DATA_BLOCK "iPar_Data_Bridge"	// DB 1920
TITLE = Vorlage Datenbaustein zur Ablage der iParameter für FB37
//Template data block used in combination with FB37
//
AUTHOR : JPR
FAMILY : WAGOiPar
NAME : iParUDL4
VERSION : 5.1
  STRUCT
   versionInfo_1 : INT  := 37;	//version info main
   versionInfo_2 : WORD  := W#16#501;	//version info release
   chkInfoData : WORD ;	//check info data
   fctReqTimeout : INT  := 6000;	//function request timeout (default 6000; av.cycle plc 5 ms - timeout 30 s)
   maxModules : INT  := 1;	//amount PROFIsafe modules FB41
   type_module_1 : INT ;	//type module 1 (661/662/663/666/667/669)
   adr_module_1 : INT ;	//I/O address module 1
   bussystem_mod_1 : INT ;	//used bussystem module 1 (0 = DP / 1 = PN)
   type_module_2 : INT ;	//type module 2 (661/662/663/666/667/669)
   adr_module_2 : INT ;	//I/O address module 2
   bussystem_mod_2 : INT ;	//used bussystem module 2 (0 = DP / 1 = PN)
   type_module_3 : INT ;	//type module 3 (661/662/663/666/667/669)
   adr_module_3 : INT ;	//I/O address module 3
   bussystem_mod_3 : INT ;	//used bussystem module 3 (0 = DP / 1 = PN)
   type_module_4 : INT ;	//type module 4 (661/662/663/666/667/669)
   adr_module_4 : INT ;	//I/O address module 4
   bussystem_mod_4 : INT ;	//used bussystem module 4 (0 = DP / 1 = PN)
   spare_34 : WORD ;
   spare_36 : WORD ;
   spare_38 : WORD ;
   spare_40 : WORD ;
   spare_42 : WORD ;
   spare_44 : WORD ;
   spare_46 : WORD ;
   spare_48 : WORD ;
   spare_50 : WORD ;
   spare_52 : WORD ;
   spare_54 : WORD ;
   spare_56 : WORD ;
   spare_58 : WORD ;
   spare_60 : WORD ;
   spare_62 : WORD ;
   spare_64 : WORD ;
   spare_66 : WORD ;
   spare_68 : WORD ;
   spare_70 : WORD ;
   spare_72 : WORD ;
   spare_74 : WORD ;
   spare_76 : WORD ;
   spare_78 : WORD ;
   spare_80 : WORD ;
   resFctReq_ok : DWORD ;	//response function request ok - "bit per module"
   resFctReq_error : DWORD ;	//response function request error - "bit per module"
   startupDate : DATE ;	//startup date application slave
   startupTime : TIME_OF_DAY ;	//startup time application slave
   slaveConfigInfo : DWORD ;	//info available PROFIsafe modules at slave
   QBAD_moduleActive : DWORD ;	//info QBAD at PROFIsafe module active
   ACK_REQ_moduleActive : DWORD ;	//info ACK_REQ at PROFIsafe module active
   READ_DIAG_REQ_module : DWORD ;	//info READ_DIAG_REQ at PROFIsafe module active
   init_fb_done : DWORD ;	//info init FB done
   check_cfg_done : DWORD ;	//info check cfg done
   upload_done : DWORD ;	//info upload slave done
   download_done : DWORD ;	//info download slave done
   compare_done : DWORD ;	//info compare slave done
   actDateCyle : DATE ;	//actual system date of cycle
   actTimeCyle : TIME_OF_DAY ;	//actual system time of cycle
   cmdCtrl_FB37 : WORD ;	//cmd / ctrl information FB37
   comCountStart_1 : WORD ;	//comCountStart indication 1
   mod_type_1 : WORD ;	//module type 1
   mod_version_1 : WORD ;	//module version 1
   spare_146 : WORD ;
   spare_148 : WORD ;
   upl_date_mod_1 : DATE ;	//upload date module 1
   upl_time_mod_1 : TIME_OF_DAY ;	//upload time module 1
   dnl_date_mod_1 : DATE ;	//download date module 1
   dnl_time_mod_1 : TIME_OF_DAY ;	//download time module 1
   cmp_date_mod_1 : DATE ;	//compare date module 1
   cmp_time_mod_1 : TIME_OF_DAY ;	//compare time module 1
   dsv_info_mod_1 : WORD ;	//dataset info module 1
   data_0_mod_1 : WORD ;	//data 0 - 1 module 1
   data_2_mod_1 : WORD ;	//data 2 - 3 module 1
   data_4_mod_1 : WORD ;	//data 4 - 5 module 1
   data_6_mod_1 : WORD ;	//data 6 - 7 module 1
   data_8_mod_1 : WORD ;	//data 8 - 9 module 1
   data_10_mod_1 : WORD ;	//data 10 - 11 module 1
   data_12_mod_1 : WORD ;	//data 12 - 13 module 1
   data_14_mod_1 : WORD ;	//data 14 - 15 module 1
   data_16_mod_1 : WORD ;	//data 16 - 17 module 1
   data_18_mod_1 : WORD ;	//data 18 - 19 module 1
   data_20_mod_1 : WORD ;	//data 20 - 21 module 1
   data_22_mod_1 : WORD ;	//data 22 - 23 module 1
   data_24_mod_1 : WORD ;	//data 24 - 25 module 1
   data_26_mod_1 : WORD ;	//data 26 - 27 module 1
   data_28_mod_1 : WORD ;	//data 28 - 29 module 1
   data_30_mod_1 : WORD ;	//data 30 - 31 module 1
   data_32_mod_1 : WORD ;	//data 32 - 33 module 1
   data_34_mod_1 : WORD ;	//data 34 - 35 module 1
   data_36_mod_1 : WORD ;	//data 36 - 37 module 1
   data_38_mod_1 : WORD ;	//data 38 - 39 module 1
   spare_210 : WORD ;
   spare_212 : WORD ;
   spare_214 : WORD ;
   spare_216 : WORD ;
   spare_218 : WORD ;
   error_Com_1 : WORD ;	//error indication  Com  module 1
   error_nb_Com_1 : WORD ;	//error number indication  Com  module 1
   state_SFB52a_1 : WORD ;	//state SFB52 part 1 module 1
   state_SFB52b_1 : WORD ;	//state SFB52 part 2 module 1
   state_SFB53a_1 : WORD ;	//state SFB53 part 1 module 1
   state_SFB53b_1 : WORD ;	//state SFB53 part 2 module 1
   spare_232 : WORD ;
   error_date_mod_1 : DATE ;	//error date module 1
   error_time_mod_1 : TIME_OF_DAY ;	//error time module 1
   error_info_mod_1 : WORD ;	//error info read values module 1
   error_F_Module_mod_1 : WORD ;	//error safety module module 1
   error_F_DI_1_mod_1 : WORD ;	//error safety input 1 module 1
   error_F_DI_2_mod_1 : WORD ;	//error safety input 2 module 1
   error_F_DI_3_mod_1 : WORD ;	//error safety input 3 module 1
   error_F_DI_4_mod_1 : WORD ;	//error safety input 4 module 1
   error_F_DI_5_mod_1 : WORD ;	//error safety input 5 module 1
   error_F_DI_6_mod_1 : WORD ;	//error safety input 6 module 1
   error_F_DI_7_mod_1 : WORD ;	//error safety input 7 module 1
   error_F_DI_8_mod_1 : WORD ;	//error safety input 8 module 1
   error_F_DO_1_mod_1 : WORD ;	//error safety output 1 module 1
   error_F_DO_2_mod_1 : WORD ;	//error safety output 2 module 1
   error_F_DO_3_mod_1 : WORD ;	//error safety output 3 module 1
   error_F_DO_4_mod_1 : WORD ;	//error safety output 4 module 1
   error_Reg52_mod_1 : WORD ;	//error safety module register 52 module 1
   error_Reg53_mod_1 : WORD ;	//error safety module register 53 module 1
   error_Reg54_mod_1 : WORD ;	//error safety module register 54 module 1
   error_Reg55_mod_1 : WORD ;	//error safety module register 55 module 1
   spare_276 : WORD ;
   spare_278 : WORD ;
   comCountStart_2 : WORD ;	//comCountStart indication 2
   mod_type_2 : WORD ;	//module type 2
   mod_version_2 : WORD ;	//module version 2
   spare_286 : WORD ;
   spare_288 : WORD ;
   upl_date_mod_2 : DATE ;	//upload date module 2
   upl_time_mod_2 : TIME_OF_DAY ;	//upload time module 2
   dnl_date_mod_2 : DATE ;	//download date module 2
   dnl_time_mod_2 : TIME_OF_DAY ;	//download time module 2
   cmp_date_mod_2 : DATE ;	//compare date module 2
   cmp_time_mod_2 : TIME_OF_DAY ;	//compare time module 2
   dsv_info_mod_2 : WORD ;	//dataset info module 2
   data_0_mod_2 : WORD ;	//data 0 - 1 module 2
   data_2_mod_2 : WORD ;	//data 2 - 3 module 2
   data_4_mod_2 : WORD ;	//data 4 - 5 module 2
   data_6_mod_2 : WORD ;	//data 6 - 7 module 2
   data_8_mod_2 : WORD ;	//data 8 - 9 module 2
   data_10_mod_2 : WORD ;	//data 10 - 11 module 2
   data_12_mod_2 : WORD ;	//data 12 - 13 module 2
   data_14_mod_2 : WORD ;	//data 14 - 15 module 2
   data_16_mod_2 : WORD ;	//data 16 - 17 module 2
   data_18_mod_2 : WORD ;	//data 18 - 19 module 2
   data_20_mod_2 : WORD ;	//data 20 - 21 module 2
   data_22_mod_2 : WORD ;	//data 22 - 23 module 2
   data_24_mod_2 : WORD ;	//data 24 - 25 module 2
   data_26_mod_2 : WORD ;	//data 26 - 27 module 2
   data_28_mod_2 : WORD ;	//data 28 - 29 module 2
   data_30_mod_2 : WORD ;	//data 30 - 31 module 2
   data_32_mod_2 : WORD ;	//data 32 - 33 module 2
   data_34_mod_2 : WORD ;	//data 34 - 35 module 2
   data_36_mod_2 : WORD ;	//data 36 - 37 module 2
   data_38_mod_2 : WORD ;	//data 38 - 39 module 2
   spare_350 : WORD ;
   spare_352 : WORD ;
   spare_354 : WORD ;
   spare_356 : WORD ;
   spare_358 : WORD ;
   error_Com_2 : WORD ;	//error indication  Com  module 2
   error_nb_Com_2 : WORD ;	//error number indication  Com  module 2
   state_SFB52a_2 : WORD ;	//state SFB52 part 1 module 2
   state_SFB52b_2 : WORD ;	//state SFB52 part 2 module 2
   state_SFB53a_2 : WORD ;	//state SFB53 part 1 module 2
   state_SFB53b_2 : WORD ;	//state SFB53 part 2 module 2
   spare_372 : WORD ;
   error_date_mod_2 : DATE ;	//error date module 2
   error_time_mod_2 : TIME_OF_DAY ;	//error time module 2
   error_info_mod_2 : WORD ;	//error info read values module 2
   error_F_Module_mod_2 : WORD ;	//error safety module module 2
   error_F_DI_1_mod_2 : WORD ;	//error safety input 1 module 2
   error_F_DI_2_mod_2 : WORD ;	//error safety input 2 module 2
   error_F_DI_3_mod_2 : WORD ;	//error safety input 3 module 2
   error_F_DI_4_mod_2 : WORD ;	//error safety input 4 module 2
   error_F_DI_5_mod_2 : WORD ;	//error safety input 5 module 2
   error_F_DI_6_mod_2 : WORD ;	//error safety input 6 module 2
   error_F_DI_7_mod_2 : WORD ;	//error safety input 7 module 2
   error_F_DI_8_mod_2 : WORD ;	//error safety input 8 module 2
   error_F_DO_1_mod_2 : WORD ;	//error safety output 1 module 2
   error_F_DO_2_mod_2 : WORD ;	//error safety output 2 module 2
   error_F_DO_3_mod_2 : WORD ;	//error safety output 3 module 2
   error_F_DO_4_mod_2 : WORD ;	//error safety output 4 module 2
   error_Reg52_mod_2 : WORD ;	//error safety module register 52 module 2
   error_Reg53_mod_2 : WORD ;	//error safety module register 53 module 2
   error_Reg54_mod_2 : WORD ;	//error safety module register 54 module 2
   error_Reg55_mod_2 : WORD ;	//error safety module register 55 module 2
   spare_416 : WORD ;
   spare_418 : WORD ;
   comCountStart_3 : WORD ;	//comCountStart indication 3
   mod_type_3 : WORD ;	//module type 3
   mod_version_3 : WORD ;	//module version 3
   spare_426 : WORD ;
   spare_428 : WORD ;
   upl_date_mod_3 : DATE ;	//upload date module 3
   upl_time_mod_3 : TIME_OF_DAY ;	//upload time module 3
   dnl_date_mod_3 : DATE ;	//download date module 3
   dnl_time_mod_3 : TIME_OF_DAY ;	//download time module 3
   cmp_date_mod_3 : DATE ;	//compare date module  3
   cmp_time_mod_3 : TIME_OF_DAY ;	//compare time module  3
   dsv_info_mod_3 : WORD ;	//dataset info module 3
   data_0_mod_3 : WORD ;	//data 0 - 1 module 3
   data_2_mod_3 : WORD ;	//data 2 - 3 module 3
   data_4_mod_3 : WORD ;	//data 4 - 5 module 3
   data_6_mod_3 : WORD ;	//data 6 - 7 module 3
   data_8_mod_3 : WORD ;	//data 8 - 9 module 3
   data_10_mod_3 : WORD ;	//data 10 - 11 module 3
   data_12_mod_3 : WORD ;	//data 12 - 13 module 3
   data_14_mod_3 : WORD ;	//data 14 - 15 module 3
   data_16_mod_3 : WORD ;	//data 16 - 17 module 3
   data_18_mod_3 : WORD ;	//data 18 - 19 module 3
   data_20_mod_3 : WORD ;	//data 20 - 21 module 3
   data_22_mod_3 : WORD ;	//data 22 - 23 module 3
   data_24_mod_3 : WORD ;	//data 24 - 25 module 3
   data_26_mod_3 : WORD ;	//data 26 - 27 module 3
   data_28_mod_3 : WORD ;	//data 28 - 29 module 3
   data_30_mod_3 : WORD ;	//data 30 - 31 module 3
   data_32_mod_3 : WORD ;	//data 32 - 33 module 3
   data_34_mod_3 : WORD ;	//data 34 - 35 module 3
   data_36_mod_3 : WORD ;	//data 36 - 37 module 3
   data_38_mod_3 : WORD ;	//data 38 - 39 module 3
   spare_490 : WORD ;
   spare_492 : WORD ;
   spare_494 : WORD ;
   spare_496 : WORD ;
   spare_498 : WORD ;
   error_Com_3 : WORD ;	//error indication  Com  module 3
   error_nb_Com_3 : WORD ;	//error number indication  Com  module 3
   state_SFB52a_3 : WORD ;	//state SFB52 part 1 module 3
   state_SFB52b_3 : WORD ;	//state SFB52 part 2 module 3
   state_SFB53a_3 : WORD ;	//state SFB53 part 1 module 3
   state_SFB53b_3 : WORD ;	//state SFB53 part 2 module 3
   spare_512 : WORD ;
   error_date_mod_3 : DATE ;	//error date module 3
   error_time_mod_3 : TIME_OF_DAY ;	//error time module 3
   error_info_mod_3 : WORD ;	//error info read values module 3
   error_F_Module_mod_3 : WORD ;	//error safety module module 3
   error_F_DI_1_mod_3 : WORD ;	//error safety input 1 module 3
   error_F_DI_2_mod_3 : WORD ;	//error safety input 2 module 3
   error_F_DI_3_mod_3 : WORD ;	//error safety input 3 module 3
   error_F_DI_4_mod_3 : WORD ;	//error safety input 4 module 3
   error_F_DI_5_mod_3 : WORD ;	//error safety input 5 module 3
   error_F_DI_6_mod_3 : WORD ;	//error safety input 6 module 3
   error_F_DI_7_mod_3 : WORD ;	//error safety input 7 module 3
   error_F_DI_8_mod_3 : WORD ;	//error safety input 8 module 3
   error_F_DO_1_mod_3 : WORD ;	//error safety output 1 module 3
   error_F_DO_2_mod_3 : WORD ;	//error safety output 2 module 3
   error_F_DO_3_mod_3 : WORD ;	//error safety output 3 module 3
   error_F_DO_4_mod_3 : WORD ;	//error safety output 4 module 3
   error_Reg52_mod_3 : WORD ;	//error safety module register 52 module 3
   error_Reg53_mod_3 : WORD ;	//error safety module register 53 module 3
   error_Reg54_mod_3 : WORD ;	//error safety module register 54 module 3
   error_Reg55_mod_3 : WORD ;	//error safety module register 55 module 3
   spare_556 : WORD ;
   spare_558 : WORD ;
   comCountStart_4 : WORD ;	//comCountStart indication 4
   mod_type_4 : WORD ;	//module type  4
   mod_version_4 : WORD ;	//module version  4
   spare_566 : WORD ;
   spare_568 : WORD ;
   upl_date_mod_4 : DATE ;	//upload date module  4
   upl_time_mod_4 : TIME_OF_DAY ;	//upload time module  4
   dnl_date_mod_4 : DATE ;	//download date module  4
   dnl_time_mod_4 : TIME_OF_DAY ;	//download time module  4
   cmp_date_mod_4 : DATE ;	//compare date module   4
   cmp_time_mod_4 : TIME_OF_DAY ;	//compare time module   4
   dsv_info_mod_4 : WORD ;	//dataset info module 4
   data_0_mod_4 : WORD ;	//data 0 - 1 module  4
   data_2_mod_4 : WORD ;	//data 2 - 3 module  4
   data_4_mod_4 : WORD ;	//data 4 - 5 module  4
   data_6_mod_4 : WORD ;	//data 6 - 7 module  4
   data_8_mod_4 : WORD ;	//data 8 - 9 module  4
   data_10_mod_4 : WORD ;	//data 10 - 11 module  4
   data_12_mod_4 : WORD ;	//data 12 - 13 module  4
   data_14_mod_4 : WORD ;	//data 14 - 15 module  4
   data_16_mod_4 : WORD ;	//data 16 - 17 module  4
   data_18_mod_4 : WORD ;	//data 18 - 19 module  4
   data_20_mod_4 : WORD ;	//data 20 - 21 module  4
   data_22_mod_4 : WORD ;	//data 22 - 23 module  4
   data_24_mod_4 : WORD ;	//data 24 - 25 module  4
   data_26_mod_4 : WORD ;	//data 26 - 27 module  4
   data_28_mod_4 : WORD ;	//data 28 - 29 module  4
   data_30_mod_4 : WORD ;	//data 30 - 31 module  4
   data_32_mod_4 : WORD ;	//data 32 - 33 module  4
   data_34_mod_4 : WORD ;	//data 34 - 35 module  4
   data_36_mod_4 : WORD ;	//data 36 - 37 module  4
   data_38_mod_4 : WORD ;	//data 38 - 39 module  4
   spare_630 : WORD ;
   spare_632 : WORD ;
   spare_634 : WORD ;
   spare_636 : WORD ;
   spare_638 : WORD ;
   error_Com_4 : WORD ;	//error indication  Com  module 4
   error_nb_Com_4 : WORD ;	//error number indication  Com  module 4
   state_SFB52a_4 : WORD ;	//state SFB52 part 1 module 4
   state_SFB52b_4 : WORD ;	//state SFB52 part 2 module 4
   state_SFB53a_4 : WORD ;	//state SFB53 part 1 module 4
   state_SFB53b_4 : WORD ;	//state SFB53 part 2 module 4
   spare_652 : WORD ;
   error_date_mod_4 : DATE ;	//error date module 4
   error_time_mod_4 : TIME_OF_DAY ;	//error time module 4
   error_info_mod_4 : WORD ;	//error info read values module 4
   error_F_Module_mod_4 : WORD ;	//error safety module module 4
   error_F_DI_1_mod_4 : WORD ;	//error safety input 1 module 4
   error_F_DI_2_mod_4 : WORD ;	//error safety input 2 module 4
   error_F_DI_3_mod_4 : WORD ;	//error safety input 3 module 4
   error_F_DI_4_mod_4 : WORD ;	//error safety input 4 module 4
   error_F_DI_5_mod_4 : WORD ;	//error safety input 5 module 4
   error_F_DI_6_mod_4 : WORD ;	//error safety input 6 module 4
   error_F_DI_7_mod_4 : WORD ;	//error safety input 7 module 4
   error_F_DI_8_mod_4 : WORD ;	//error safety input 8 module 4
   error_F_DO_1_mod_4 : WORD ;	//error safety output 1 module 4
   error_F_DO_2_mod_4 : WORD ;	//error safety output 2 module 4
   error_F_DO_3_mod_4 : WORD ;	//error safety output 3 module 4
   error_F_DO_4_mod_4 : WORD ;	//error safety output 4 module 4
   error_Reg52_mod_4 : WORD ;	//error safety module register 52 module 4
   error_Reg53_mod_4 : WORD ;	//error safety module register 53 module 4
   error_Reg54_mod_4 : WORD ;	//error safety module register 54 module 4
   error_Reg55_mod_4 : WORD ;	//error safety module register 55 module 4
   spare_696 : WORD ;
   spare_698 : WORD ;
  END_STRUCT ;	
BEGIN
   versionInfo_1 := 37;
   versionInfo_2 := W#16#501;
   chkInfoData := W#16#3;
   fctReqTimeout := 6000;
   maxModules := 3;
   type_module_1 := 662;
   adr_module_1 := 40;
   bussystem_mod_1 := 1;
   type_module_2 := 667;
   adr_module_2 := 45;
   bussystem_mod_2 := 1;
   type_module_3 := 666;
   adr_module_3 := 50;
   bussystem_mod_3 := 1;
   bussystem_mod_4 := 1;
   slaveConfigInfo := DW#16#7;
   init_fb_done := DW#16#7;
   check_cfg_done := DW#16#7;
   upload_done := DW#16#7;
   download_done := DW#16#7;
   compare_done := DW#16#7;
   cmdCtrl_FB37 := W#16#FE00;
   comCountStart_1 := W#16#2;
   mod_type_1 := W#16#19E5;
   mod_version_1 := W#16#3;
   dsv_info_mod_1 := W#16#1FF0;
   data_0_mod_1 := W#16#4545;
   data_2_mod_1 := W#16#10CC;
   data_4_mod_1 := W#16#20CC;
   data_6_mod_1 := W#16#202;
   data_8_mod_1 := W#16#4FF;
   data_10_mod_1 := W#16#F;
   data_12_mod_1 := W#16#6400;
   data_14_mod_1 := W#16#6400;
   data_16_mod_1 := W#16#6400;
   data_18_mod_1 := W#16#6400;
   data_22_mod_1 := W#16#F01F;
   data_24_mod_1 := W#16#FEFF;
   data_26_mod_1 := W#16#1C72;
   data_28_mod_1 := W#16#5B54;
   data_32_mod_1 := W#16#3341;
   comCountStart_2 := W#16#2;
   mod_type_2 := W#16#1A17;
   mod_version_2 := W#16#3;
   dsv_info_mod_2 := W#16#7573;
   data_0_mod_2 := W#16#4545;
   data_2_mod_2 := W#16#10CC;
   data_4_mod_2 := W#16#20CC;
   data_6_mod_2 := W#16#203;
   data_8_mod_2 := W#16#F430;
   data_10_mod_2 := W#16#6400;
   data_12_mod_2 := W#16#6400;
   data_16_mod_2 := W#16#100;
   data_18_mod_2 := W#16#3733;
   data_20_mod_2 := W#16#7375;
   data_22_mod_2 := W#16#FEFF;
   data_24_mod_2 := W#16#B6E;
   data_26_mod_2 := W#16#5B54;
   data_30_mod_2 := W#16#7E16;
   comCountStart_3 := W#16#2;
   mod_type_3 := W#16#1A0D;
   mod_version_3 := W#16#3;
   dsv_info_mod_3 := W#16#B395;
   data_0_mod_3 := W#16#4545;
   data_2_mod_3 := W#16#10CC;
   data_4_mod_3 := W#16#20CC;
   data_6_mod_3 := W#16#204;
   data_8_mod_3 := W#16#F430;
   data_10_mod_3 := W#16#6400;
   data_12_mod_3 := W#16#6400;
   data_18_mod_3 := W#16#AA00;
   data_20_mod_3 := W#16#95B3;
   data_22_mod_3 := W#16#FEFF;
   data_24_mod_3 := W#16#CC3D;
   data_26_mod_3 := W#16#1256;
   data_30_mod_3 := W#16#E0D;
END_DATA_BLOCK

DATA_BLOCK "iPar_Data_Trolley"	// DB 1921
TITLE = Vorlage Datenbaustein zur Ablage der iParameter für FB37
//Template data block used in combination with FB37
//
AUTHOR : JPR
FAMILY : WAGOiPar
NAME : iParUDL4
VERSION : 5.1
  STRUCT
   versionInfo_1 : INT  := 37;	//version info main
   versionInfo_2 : WORD  := W#16#501;	//version info release
   chkInfoData : WORD ;	//check info data
   fctReqTimeout : INT  := 6000;	//function request timeout (default 6000; av.cycle plc 5 ms - timeout 30 s)
   maxModules : INT  := 1;	//amount PROFIsafe modules FB41
   type_module_1 : INT ;	//type module 1 (661/662/663/666/667/669)
   adr_module_1 : INT ;	//I/O address module 1
   bussystem_mod_1 : INT ;	//used bussystem module 1 (0 = DP / 1 = PN)
   type_module_2 : INT ;	//type module 2 (661/662/663/666/667/669)
   adr_module_2 : INT ;	//I/O address module 2
   bussystem_mod_2 : INT ;	//used bussystem module 2 (0 = DP / 1 = PN)
   type_module_3 : INT ;	//type module 3 (661/662/663/666/667/669)
   adr_module_3 : INT ;	//I/O address module 3
   bussystem_mod_3 : INT ;	//used bussystem module 3 (0 = DP / 1 = PN)
   type_module_4 : INT ;	//type module 4 (661/662/663/666/667/669)
   adr_module_4 : INT ;	//I/O address module 4
   bussystem_mod_4 : INT ;	//used bussystem module 4 (0 = DP / 1 = PN)
   spare_34 : WORD ;
   spare_36 : WORD ;
   spare_38 : WORD ;
   spare_40 : WORD ;
   spare_42 : WORD ;
   spare_44 : WORD ;
   spare_46 : WORD ;
   spare_48 : WORD ;
   spare_50 : WORD ;
   spare_52 : WORD ;
   spare_54 : WORD ;
   spare_56 : WORD ;
   spare_58 : WORD ;
   spare_60 : WORD ;
   spare_62 : WORD ;
   spare_64 : WORD ;
   spare_66 : WORD ;
   spare_68 : WORD ;
   spare_70 : WORD ;
   spare_72 : WORD ;
   spare_74 : WORD ;
   spare_76 : WORD ;
   spare_78 : WORD ;
   spare_80 : WORD ;
   resFctReq_ok : DWORD ;	//response function request ok - "bit per module"
   resFctReq_error : DWORD ;	//response function request error - "bit per module"
   startupDate : DATE ;	//startup date application slave
   startupTime : TIME_OF_DAY ;	//startup time application slave
   slaveConfigInfo : DWORD ;	//info available PROFIsafe modules at slave
   QBAD_moduleActive : DWORD ;	//info QBAD at PROFIsafe module active
   ACK_REQ_moduleActive : DWORD ;	//info ACK_REQ at PROFIsafe module active
   READ_DIAG_REQ_module : DWORD ;	//info READ_DIAG_REQ at PROFIsafe module active
   init_fb_done : DWORD ;	//info init FB done
   check_cfg_done : DWORD ;	//info check cfg done
   upload_done : DWORD ;	//info upload slave done
   download_done : DWORD ;	//info download slave done
   compare_done : DWORD ;	//info compare slave done
   actDateCyle : DATE ;	//actual system date of cycle
   actTimeCyle : TIME_OF_DAY ;	//actual system time of cycle
   cmdCtrl_FB37 : WORD ;	//cmd / ctrl information FB37
   comCountStart_1 : WORD ;	//comCountStart indication 1
   mod_type_1 : WORD ;	//module type 1
   mod_version_1 : WORD ;	//module version 1
   spare_146 : WORD ;
   spare_148 : WORD ;
   upl_date_mod_1 : DATE ;	//upload date module 1
   upl_time_mod_1 : TIME_OF_DAY ;	//upload time module 1
   dnl_date_mod_1 : DATE ;	//download date module 1
   dnl_time_mod_1 : TIME_OF_DAY ;	//download time module 1
   cmp_date_mod_1 : DATE ;	//compare date module 1
   cmp_time_mod_1 : TIME_OF_DAY ;	//compare time module 1
   dsv_info_mod_1 : WORD ;	//dataset info module 1
   data_0_mod_1 : WORD ;	//data 0 - 1 module 1
   data_2_mod_1 : WORD ;	//data 2 - 3 module 1
   data_4_mod_1 : WORD ;	//data 4 - 5 module 1
   data_6_mod_1 : WORD ;	//data 6 - 7 module 1
   data_8_mod_1 : WORD ;	//data 8 - 9 module 1
   data_10_mod_1 : WORD ;	//data 10 - 11 module 1
   data_12_mod_1 : WORD ;	//data 12 - 13 module 1
   data_14_mod_1 : WORD ;	//data 14 - 15 module 1
   data_16_mod_1 : WORD ;	//data 16 - 17 module 1
   data_18_mod_1 : WORD ;	//data 18 - 19 module 1
   data_20_mod_1 : WORD ;	//data 20 - 21 module 1
   data_22_mod_1 : WORD ;	//data 22 - 23 module 1
   data_24_mod_1 : WORD ;	//data 24 - 25 module 1
   data_26_mod_1 : WORD ;	//data 26 - 27 module 1
   data_28_mod_1 : WORD ;	//data 28 - 29 module 1
   data_30_mod_1 : WORD ;	//data 30 - 31 module 1
   data_32_mod_1 : WORD ;	//data 32 - 33 module 1
   data_34_mod_1 : WORD ;	//data 34 - 35 module 1
   data_36_mod_1 : WORD ;	//data 36 - 37 module 1
   data_38_mod_1 : WORD ;	//data 38 - 39 module 1
   spare_210 : WORD ;
   spare_212 : WORD ;
   spare_214 : WORD ;
   spare_216 : WORD ;
   spare_218 : WORD ;
   error_Com_1 : WORD ;	//error indication  Com  module 1
   error_nb_Com_1 : WORD ;	//error number indication  Com  module 1
   state_SFB52a_1 : WORD ;	//state SFB52 part 1 module 1
   state_SFB52b_1 : WORD ;	//state SFB52 part 2 module 1
   state_SFB53a_1 : WORD ;	//state SFB53 part 1 module 1
   state_SFB53b_1 : WORD ;	//state SFB53 part 2 module 1
   spare_232 : WORD ;
   error_date_mod_1 : DATE ;	//error date module 1
   error_time_mod_1 : TIME_OF_DAY ;	//error time module 1
   error_info_mod_1 : WORD ;	//error info read values module 1
   error_F_Module_mod_1 : WORD ;	//error safety module module 1
   error_F_DI_1_mod_1 : WORD ;	//error safety input 1 module 1
   error_F_DI_2_mod_1 : WORD ;	//error safety input 2 module 1
   error_F_DI_3_mod_1 : WORD ;	//error safety input 3 module 1
   error_F_DI_4_mod_1 : WORD ;	//error safety input 4 module 1
   error_F_DI_5_mod_1 : WORD ;	//error safety input 5 module 1
   error_F_DI_6_mod_1 : WORD ;	//error safety input 6 module 1
   error_F_DI_7_mod_1 : WORD ;	//error safety input 7 module 1
   error_F_DI_8_mod_1 : WORD ;	//error safety input 8 module 1
   error_F_DO_1_mod_1 : WORD ;	//error safety output 1 module 1
   error_F_DO_2_mod_1 : WORD ;	//error safety output 2 module 1
   error_F_DO_3_mod_1 : WORD ;	//error safety output 3 module 1
   error_F_DO_4_mod_1 : WORD ;	//error safety output 4 module 1
   error_Reg52_mod_1 : WORD ;	//error safety module register 52 module 1
   error_Reg53_mod_1 : WORD ;	//error safety module register 53 module 1
   error_Reg54_mod_1 : WORD ;	//error safety module register 54 module 1
   error_Reg55_mod_1 : WORD ;	//error safety module register 55 module 1
   spare_276 : WORD ;
   spare_278 : WORD ;
   comCountStart_2 : WORD ;	//comCountStart indication 2
   mod_type_2 : WORD ;	//module type 2
   mod_version_2 : WORD ;	//module version 2
   spare_286 : WORD ;
   spare_288 : WORD ;
   upl_date_mod_2 : DATE ;	//upload date module 2
   upl_time_mod_2 : TIME_OF_DAY ;	//upload time module 2
   dnl_date_mod_2 : DATE ;	//download date module 2
   dnl_time_mod_2 : TIME_OF_DAY ;	//download time module 2
   cmp_date_mod_2 : DATE ;	//compare date module 2
   cmp_time_mod_2 : TIME_OF_DAY ;	//compare time module 2
   dsv_info_mod_2 : WORD ;	//dataset info module 2
   data_0_mod_2 : WORD ;	//data 0 - 1 module 2
   data_2_mod_2 : WORD ;	//data 2 - 3 module 2
   data_4_mod_2 : WORD ;	//data 4 - 5 module 2
   data_6_mod_2 : WORD ;	//data 6 - 7 module 2
   data_8_mod_2 : WORD ;	//data 8 - 9 module 2
   data_10_mod_2 : WORD ;	//data 10 - 11 module 2
   data_12_mod_2 : WORD ;	//data 12 - 13 module 2
   data_14_mod_2 : WORD ;	//data 14 - 15 module 2
   data_16_mod_2 : WORD ;	//data 16 - 17 module 2
   data_18_mod_2 : WORD ;	//data 18 - 19 module 2
   data_20_mod_2 : WORD ;	//data 20 - 21 module 2
   data_22_mod_2 : WORD ;	//data 22 - 23 module 2
   data_24_mod_2 : WORD ;	//data 24 - 25 module 2
   data_26_mod_2 : WORD ;	//data 26 - 27 module 2
   data_28_mod_2 : WORD ;	//data 28 - 29 module 2
   data_30_mod_2 : WORD ;	//data 30 - 31 module 2
   data_32_mod_2 : WORD ;	//data 32 - 33 module 2
   data_34_mod_2 : WORD ;	//data 34 - 35 module 2
   data_36_mod_2 : WORD ;	//data 36 - 37 module 2
   data_38_mod_2 : WORD ;	//data 38 - 39 module 2
   spare_350 : WORD ;
   spare_352 : WORD ;
   spare_354 : WORD ;
   spare_356 : WORD ;
   spare_358 : WORD ;
   error_Com_2 : WORD ;	//error indication  Com  module 2
   error_nb_Com_2 : WORD ;	//error number indication  Com  module 2
   state_SFB52a_2 : WORD ;	//state SFB52 part 1 module 2
   state_SFB52b_2 : WORD ;	//state SFB52 part 2 module 2
   state_SFB53a_2 : WORD ;	//state SFB53 part 1 module 2
   state_SFB53b_2 : WORD ;	//state SFB53 part 2 module 2
   spare_372 : WORD ;
   error_date_mod_2 : DATE ;	//error date module 2
   error_time_mod_2 : TIME_OF_DAY ;	//error time module 2
   error_info_mod_2 : WORD ;	//error info read values module 2
   error_F_Module_mod_2 : WORD ;	//error safety module module 2
   error_F_DI_1_mod_2 : WORD ;	//error safety input 1 module 2
   error_F_DI_2_mod_2 : WORD ;	//error safety input 2 module 2
   error_F_DI_3_mod_2 : WORD ;	//error safety input 3 module 2
   error_F_DI_4_mod_2 : WORD ;	//error safety input 4 module 2
   error_F_DI_5_mod_2 : WORD ;	//error safety input 5 module 2
   error_F_DI_6_mod_2 : WORD ;	//error safety input 6 module 2
   error_F_DI_7_mod_2 : WORD ;	//error safety input 7 module 2
   error_F_DI_8_mod_2 : WORD ;	//error safety input 8 module 2
   error_F_DO_1_mod_2 : WORD ;	//error safety output 1 module 2
   error_F_DO_2_mod_2 : WORD ;	//error safety output 2 module 2
   error_F_DO_3_mod_2 : WORD ;	//error safety output 3 module 2
   error_F_DO_4_mod_2 : WORD ;	//error safety output 4 module 2
   error_Reg52_mod_2 : WORD ;	//error safety module register 52 module 2
   error_Reg53_mod_2 : WORD ;	//error safety module register 53 module 2
   error_Reg54_mod_2 : WORD ;	//error safety module register 54 module 2
   error_Reg55_mod_2 : WORD ;	//error safety module register 55 module 2
   spare_416 : WORD ;
   spare_418 : WORD ;
   comCountStart_3 : WORD ;	//comCountStart indication 3
   mod_type_3 : WORD ;	//module type 3
   mod_version_3 : WORD ;	//module version 3
   spare_426 : WORD ;
   spare_428 : WORD ;
   upl_date_mod_3 : DATE ;	//upload date module 3
   upl_time_mod_3 : TIME_OF_DAY ;	//upload time module 3
   dnl_date_mod_3 : DATE ;	//download date module 3
   dnl_time_mod_3 : TIME_OF_DAY ;	//download time module 3
   cmp_date_mod_3 : DATE ;	//compare date module  3
   cmp_time_mod_3 : TIME_OF_DAY ;	//compare time module  3
   dsv_info_mod_3 : WORD ;	//dataset info module 3
   data_0_mod_3 : WORD ;	//data 0 - 1 module 3
   data_2_mod_3 : WORD ;	//data 2 - 3 module 3
   data_4_mod_3 : WORD ;	//data 4 - 5 module 3
   data_6_mod_3 : WORD ;	//data 6 - 7 module 3
   data_8_mod_3 : WORD ;	//data 8 - 9 module 3
   data_10_mod_3 : WORD ;	//data 10 - 11 module 3
   data_12_mod_3 : WORD ;	//data 12 - 13 module 3
   data_14_mod_3 : WORD ;	//data 14 - 15 module 3
   data_16_mod_3 : WORD ;	//data 16 - 17 module 3
   data_18_mod_3 : WORD ;	//data 18 - 19 module 3
   data_20_mod_3 : WORD ;	//data 20 - 21 module 3
   data_22_mod_3 : WORD ;	//data 22 - 23 module 3
   data_24_mod_3 : WORD ;	//data 24 - 25 module 3
   data_26_mod_3 : WORD ;	//data 26 - 27 module 3
   data_28_mod_3 : WORD ;	//data 28 - 29 module 3
   data_30_mod_3 : WORD ;	//data 30 - 31 module 3
   data_32_mod_3 : WORD ;	//data 32 - 33 module 3
   data_34_mod_3 : WORD ;	//data 34 - 35 module 3
   data_36_mod_3 : WORD ;	//data 36 - 37 module 3
   data_38_mod_3 : WORD ;	//data 38 - 39 module 3
   spare_490 : WORD ;
   spare_492 : WORD ;
   spare_494 : WORD ;
   spare_496 : WORD ;
   spare_498 : WORD ;
   error_Com_3 : WORD ;	//error indication  Com  module 3
   error_nb_Com_3 : WORD ;	//error number indication  Com  module 3
   state_SFB52a_3 : WORD ;	//state SFB52 part 1 module 3
   state_SFB52b_3 : WORD ;	//state SFB52 part 2 module 3
   state_SFB53a_3 : WORD ;	//state SFB53 part 1 module 3
   state_SFB53b_3 : WORD ;	//state SFB53 part 2 module 3
   spare_512 : WORD ;
   error_date_mod_3 : DATE ;	//error date module 3
   error_time_mod_3 : TIME_OF_DAY ;	//error time module 3
   error_info_mod_3 : WORD ;	//error info read values module 3
   error_F_Module_mod_3 : WORD ;	//error safety module module 3
   error_F_DI_1_mod_3 : WORD ;	//error safety input 1 module 3
   error_F_DI_2_mod_3 : WORD ;	//error safety input 2 module 3
   error_F_DI_3_mod_3 : WORD ;	//error safety input 3 module 3
   error_F_DI_4_mod_3 : WORD ;	//error safety input 4 module 3
   error_F_DI_5_mod_3 : WORD ;	//error safety input 5 module 3
   error_F_DI_6_mod_3 : WORD ;	//error safety input 6 module 3
   error_F_DI_7_mod_3 : WORD ;	//error safety input 7 module 3
   error_F_DI_8_mod_3 : WORD ;	//error safety input 8 module 3
   error_F_DO_1_mod_3 : WORD ;	//error safety output 1 module 3
   error_F_DO_2_mod_3 : WORD ;	//error safety output 2 module 3
   error_F_DO_3_mod_3 : WORD ;	//error safety output 3 module 3
   error_F_DO_4_mod_3 : WORD ;	//error safety output 4 module 3
   error_Reg52_mod_3 : WORD ;	//error safety module register 52 module 3
   error_Reg53_mod_3 : WORD ;	//error safety module register 53 module 3
   error_Reg54_mod_3 : WORD ;	//error safety module register 54 module 3
   error_Reg55_mod_3 : WORD ;	//error safety module register 55 module 3
   spare_556 : WORD ;
   spare_558 : WORD ;
   comCountStart_4 : WORD ;	//comCountStart indication 4
   mod_type_4 : WORD ;	//module type  4
   mod_version_4 : WORD ;	//module version  4
   spare_566 : WORD ;
   spare_568 : WORD ;
   upl_date_mod_4 : DATE ;	//upload date module  4
   upl_time_mod_4 : TIME_OF_DAY ;	//upload time module  4
   dnl_date_mod_4 : DATE ;	//download date module  4
   dnl_time_mod_4 : TIME_OF_DAY ;	//download time module  4
   cmp_date_mod_4 : DATE ;	//compare date module   4
   cmp_time_mod_4 : TIME_OF_DAY ;	//compare time module   4
   dsv_info_mod_4 : WORD ;	//dataset info module 4
   data_0_mod_4 : WORD ;	//data 0 - 1 module  4
   data_2_mod_4 : WORD ;	//data 2 - 3 module  4
   data_4_mod_4 : WORD ;	//data 4 - 5 module  4
   data_6_mod_4 : WORD ;	//data 6 - 7 module  4
   data_8_mod_4 : WORD ;	//data 8 - 9 module  4
   data_10_mod_4 : WORD ;	//data 10 - 11 module  4
   data_12_mod_4 : WORD ;	//data 12 - 13 module  4
   data_14_mod_4 : WORD ;	//data 14 - 15 module  4
   data_16_mod_4 : WORD ;	//data 16 - 17 module  4
   data_18_mod_4 : WORD ;	//data 18 - 19 module  4
   data_20_mod_4 : WORD ;	//data 20 - 21 module  4
   data_22_mod_4 : WORD ;	//data 22 - 23 module  4
   data_24_mod_4 : WORD ;	//data 24 - 25 module  4
   data_26_mod_4 : WORD ;	//data 26 - 27 module  4
   data_28_mod_4 : WORD ;	//data 28 - 29 module  4
   data_30_mod_4 : WORD ;	//data 30 - 31 module  4
   data_32_mod_4 : WORD ;	//data 32 - 33 module  4
   data_34_mod_4 : WORD ;	//data 34 - 35 module  4
   data_36_mod_4 : WORD ;	//data 36 - 37 module  4
   data_38_mod_4 : WORD ;	//data 38 - 39 module  4
   spare_630 : WORD ;
   spare_632 : WORD ;
   spare_634 : WORD ;
   spare_636 : WORD ;
   spare_638 : WORD ;
   error_Com_4 : WORD ;	//error indication  Com  module 4
   error_nb_Com_4 : WORD ;	//error number indication  Com  module 4
   state_SFB52a_4 : WORD ;	//state SFB52 part 1 module 4
   state_SFB52b_4 : WORD ;	//state SFB52 part 2 module 4
   state_SFB53a_4 : WORD ;	//state SFB53 part 1 module 4
   state_SFB53b_4 : WORD ;	//state SFB53 part 2 module 4
   spare_652 : WORD ;
   error_date_mod_4 : DATE ;	//error date module 4
   error_time_mod_4 : TIME_OF_DAY ;	//error time module 4
   error_info_mod_4 : WORD ;	//error info read values module 4
   error_F_Module_mod_4 : WORD ;	//error safety module module 4
   error_F_DI_1_mod_4 : WORD ;	//error safety input 1 module 4
   error_F_DI_2_mod_4 : WORD ;	//error safety input 2 module 4
   error_F_DI_3_mod_4 : WORD ;	//error safety input 3 module 4
   error_F_DI_4_mod_4 : WORD ;	//error safety input 4 module 4
   error_F_DI_5_mod_4 : WORD ;	//error safety input 5 module 4
   error_F_DI_6_mod_4 : WORD ;	//error safety input 6 module 4
   error_F_DI_7_mod_4 : WORD ;	//error safety input 7 module 4
   error_F_DI_8_mod_4 : WORD ;	//error safety input 8 module 4
   error_F_DO_1_mod_4 : WORD ;	//error safety output 1 module 4
   error_F_DO_2_mod_4 : WORD ;	//error safety output 2 module 4
   error_F_DO_3_mod_4 : WORD ;	//error safety output 3 module 4
   error_F_DO_4_mod_4 : WORD ;	//error safety output 4 module 4
   error_Reg52_mod_4 : WORD ;	//error safety module register 52 module 4
   error_Reg53_mod_4 : WORD ;	//error safety module register 53 module 4
   error_Reg54_mod_4 : WORD ;	//error safety module register 54 module 4
   error_Reg55_mod_4 : WORD ;	//error safety module register 55 module 4
   spare_696 : WORD ;
   spare_698 : WORD ;
  END_STRUCT ;	
BEGIN
   versionInfo_1 := 37;
   versionInfo_2 := W#16#501;
   chkInfoData := W#16#3;
   fctReqTimeout := 6000;
   maxModules := 3;
   type_module_1 := 667;
   adr_module_1 := 35;
   bussystem_mod_1 := 1;
   type_module_2 := 667;
   adr_module_2 := 40;
   bussystem_mod_2 := 1;
   type_module_3 := 661;
   adr_module_3 := 45;
   bussystem_mod_3 := 1;
   bussystem_mod_4 := 1;
   slaveConfigInfo := DW#16#7;
   init_fb_done := DW#16#7;
   check_cfg_done := DW#16#7;
   upload_done := DW#16#7;
   download_done := DW#16#7;
   compare_done := DW#16#7;
   cmdCtrl_FB37 := W#16#FE00;
   comCountStart_1 := W#16#2;
   mod_type_1 := W#16#1A17;
   mod_version_1 := W#16#3;
   dsv_info_mod_1 := W#16#317C;
   data_0_mod_1 := W#16#4545;
   data_2_mod_1 := W#16#10CC;
   data_4_mod_1 := W#16#20CC;
   data_6_mod_1 := W#16#203;
   data_8_mod_1 := W#16#F430;
   data_10_mod_1 := W#16#6400;
   data_12_mod_1 := W#16#6400;
   data_18_mod_1 := W#16#3333;
   data_20_mod_1 := W#16#7C31;
   data_22_mod_1 := W#16#FEFF;
   data_30_mod_1 := W#16#B7BF;
   comCountStart_2 := W#16#2;
   mod_type_2 := W#16#1A17;
   mod_version_2 := W#16#3;
   dsv_info_mod_2 := W#16#784F;
   data_0_mod_2 := W#16#4545;
   data_2_mod_2 := W#16#10CC;
   data_4_mod_2 := W#16#20CC;
   data_6_mod_2 := W#16#203;
   data_8_mod_2 := W#16#F432;
   data_10_mod_2 := W#16#6400;
   data_12_mod_2 := W#16#6400;
   data_18_mod_2 := W#16#3333;
   data_20_mod_2 := W#16#4F78;
   data_22_mod_2 := W#16#FEFF;
   data_24_mod_2 := W#16#3DF1;
   data_26_mod_2 := W#16#3D5B;
   data_30_mod_2 := W#16#E622;
   comCountStart_3 := W#16#2;
   mod_type_3 := W#16#19DB;
   mod_version_3 := W#16#3;
   dsv_info_mod_3 := W#16#A98A;
   data_0_mod_3 := W#16#4545;
   data_2_mod_3 := W#16#10CC;
   data_4_mod_3 := W#16#20CC;
   data_6_mod_3 := W#16#201;
   data_8_mod_3 := W#16#F430;
   data_10_mod_3 := W#16#6400;
   data_12_mod_3 := W#16#6400;
   data_16_mod_3 := W#16#8AA9;
   data_18_mod_3 := W#16#FEFF;
   data_26_mod_3 := W#16#A84E;
END_DATA_BLOCK

DATA_BLOCK "iPar_Data_Lift"	// DB 1922
TITLE = Vorlage Datenbaustein zur Ablage der iParameter für FB37
//Template data block used in combination with FB37
//
AUTHOR : JPR
FAMILY : WAGOiPar
NAME : iParUDL4
VERSION : 5.1
  STRUCT
   versionInfo_1 : INT  := 37;	//version info main
   versionInfo_2 : WORD  := W#16#501;	//version info release
   chkInfoData : WORD ;	//check info data
   fctReqTimeout : INT  := 6000;	//function request timeout (default 6000; av.cycle plc 5 ms - timeout 30 s)
   maxModules : INT  := 1;	//amount PROFIsafe modules FB41
   type_module_1 : INT ;	//type module 1 (661/662/663/666/667/669)
   adr_module_1 : INT ;	//I/O address module 1
   bussystem_mod_1 : INT ;	//used bussystem module 1 (0 = DP / 1 = PN)
   type_module_2 : INT ;	//type module 2 (661/662/663/666/667/669)
   adr_module_2 : INT ;	//I/O address module 2
   bussystem_mod_2 : INT ;	//used bussystem module 2 (0 = DP / 1 = PN)
   type_module_3 : INT ;	//type module 3 (661/662/663/666/667/669)
   adr_module_3 : INT ;	//I/O address module 3
   bussystem_mod_3 : INT ;	//used bussystem module 3 (0 = DP / 1 = PN)
   type_module_4 : INT ;	//type module 4 (661/662/663/666/667/669)
   adr_module_4 : INT ;	//I/O address module 4
   bussystem_mod_4 : INT ;	//used bussystem module 4 (0 = DP / 1 = PN)
   spare_34 : WORD ;
   spare_36 : WORD ;
   spare_38 : WORD ;
   spare_40 : WORD ;
   spare_42 : WORD ;
   spare_44 : WORD ;
   spare_46 : WORD ;
   spare_48 : WORD ;
   spare_50 : WORD ;
   spare_52 : WORD ;
   spare_54 : WORD ;
   spare_56 : WORD ;
   spare_58 : WORD ;
   spare_60 : WORD ;
   spare_62 : WORD ;
   spare_64 : WORD ;
   spare_66 : WORD ;
   spare_68 : WORD ;
   spare_70 : WORD ;
   spare_72 : WORD ;
   spare_74 : WORD ;
   spare_76 : WORD ;
   spare_78 : WORD ;
   spare_80 : WORD ;
   resFctReq_ok : DWORD ;	//response function request ok - "bit per module"
   resFctReq_error : DWORD ;	//response function request error - "bit per module"
   startupDate : DATE ;	//startup date application slave
   startupTime : TIME_OF_DAY ;	//startup time application slave
   slaveConfigInfo : DWORD ;	//info available PROFIsafe modules at slave
   QBAD_moduleActive : DWORD ;	//info QBAD at PROFIsafe module active
   ACK_REQ_moduleActive : DWORD ;	//info ACK_REQ at PROFIsafe module active
   READ_DIAG_REQ_module : DWORD ;	//info READ_DIAG_REQ at PROFIsafe module active
   init_fb_done : DWORD ;	//info init FB done
   check_cfg_done : DWORD ;	//info check cfg done
   upload_done : DWORD ;	//info upload slave done
   download_done : DWORD ;	//info download slave done
   compare_done : DWORD ;	//info compare slave done
   actDateCyle : DATE ;	//actual system date of cycle
   actTimeCyle : TIME_OF_DAY ;	//actual system time of cycle
   cmdCtrl_FB37 : WORD ;	//cmd / ctrl information FB37
   comCountStart_1 : WORD ;	//comCountStart indication 1
   mod_type_1 : WORD ;	//module type 1
   mod_version_1 : WORD ;	//module version 1
   spare_146 : WORD ;
   spare_148 : WORD ;
   upl_date_mod_1 : DATE ;	//upload date module 1
   upl_time_mod_1 : TIME_OF_DAY ;	//upload time module 1
   dnl_date_mod_1 : DATE ;	//download date module 1
   dnl_time_mod_1 : TIME_OF_DAY ;	//download time module 1
   cmp_date_mod_1 : DATE ;	//compare date module 1
   cmp_time_mod_1 : TIME_OF_DAY ;	//compare time module 1
   dsv_info_mod_1 : WORD ;	//dataset info module 1
   data_0_mod_1 : WORD ;	//data 0 - 1 module 1
   data_2_mod_1 : WORD ;	//data 2 - 3 module 1
   data_4_mod_1 : WORD ;	//data 4 - 5 module 1
   data_6_mod_1 : WORD ;	//data 6 - 7 module 1
   data_8_mod_1 : WORD ;	//data 8 - 9 module 1
   data_10_mod_1 : WORD ;	//data 10 - 11 module 1
   data_12_mod_1 : WORD ;	//data 12 - 13 module 1
   data_14_mod_1 : WORD ;	//data 14 - 15 module 1
   data_16_mod_1 : WORD ;	//data 16 - 17 module 1
   data_18_mod_1 : WORD ;	//data 18 - 19 module 1
   data_20_mod_1 : WORD ;	//data 20 - 21 module 1
   data_22_mod_1 : WORD ;	//data 22 - 23 module 1
   data_24_mod_1 : WORD ;	//data 24 - 25 module 1
   data_26_mod_1 : WORD ;	//data 26 - 27 module 1
   data_28_mod_1 : WORD ;	//data 28 - 29 module 1
   data_30_mod_1 : WORD ;	//data 30 - 31 module 1
   data_32_mod_1 : WORD ;	//data 32 - 33 module 1
   data_34_mod_1 : WORD ;	//data 34 - 35 module 1
   data_36_mod_1 : WORD ;	//data 36 - 37 module 1
   data_38_mod_1 : WORD ;	//data 38 - 39 module 1
   spare_210 : WORD ;
   spare_212 : WORD ;
   spare_214 : WORD ;
   spare_216 : WORD ;
   spare_218 : WORD ;
   error_Com_1 : WORD ;	//error indication  Com  module 1
   error_nb_Com_1 : WORD ;	//error number indication  Com  module 1
   state_SFB52a_1 : WORD ;	//state SFB52 part 1 module 1
   state_SFB52b_1 : WORD ;	//state SFB52 part 2 module 1
   state_SFB53a_1 : WORD ;	//state SFB53 part 1 module 1
   state_SFB53b_1 : WORD ;	//state SFB53 part 2 module 1
   spare_232 : WORD ;
   error_date_mod_1 : DATE ;	//error date module 1
   error_time_mod_1 : TIME_OF_DAY ;	//error time module 1
   error_info_mod_1 : WORD ;	//error info read values module 1
   error_F_Module_mod_1 : WORD ;	//error safety module module 1
   error_F_DI_1_mod_1 : WORD ;	//error safety input 1 module 1
   error_F_DI_2_mod_1 : WORD ;	//error safety input 2 module 1
   error_F_DI_3_mod_1 : WORD ;	//error safety input 3 module 1
   error_F_DI_4_mod_1 : WORD ;	//error safety input 4 module 1
   error_F_DI_5_mod_1 : WORD ;	//error safety input 5 module 1
   error_F_DI_6_mod_1 : WORD ;	//error safety input 6 module 1
   error_F_DI_7_mod_1 : WORD ;	//error safety input 7 module 1
   error_F_DI_8_mod_1 : WORD ;	//error safety input 8 module 1
   error_F_DO_1_mod_1 : WORD ;	//error safety output 1 module 1
   error_F_DO_2_mod_1 : WORD ;	//error safety output 2 module 1
   error_F_DO_3_mod_1 : WORD ;	//error safety output 3 module 1
   error_F_DO_4_mod_1 : WORD ;	//error safety output 4 module 1
   error_Reg52_mod_1 : WORD ;	//error safety module register 52 module 1
   error_Reg53_mod_1 : WORD ;	//error safety module register 53 module 1
   error_Reg54_mod_1 : WORD ;	//error safety module register 54 module 1
   error_Reg55_mod_1 : WORD ;	//error safety module register 55 module 1
   spare_276 : WORD ;
   spare_278 : WORD ;
   comCountStart_2 : WORD ;	//comCountStart indication 2
   mod_type_2 : WORD ;	//module type 2
   mod_version_2 : WORD ;	//module version 2
   spare_286 : WORD ;
   spare_288 : WORD ;
   upl_date_mod_2 : DATE ;	//upload date module 2
   upl_time_mod_2 : TIME_OF_DAY ;	//upload time module 2
   dnl_date_mod_2 : DATE ;	//download date module 2
   dnl_time_mod_2 : TIME_OF_DAY ;	//download time module 2
   cmp_date_mod_2 : DATE ;	//compare date module 2
   cmp_time_mod_2 : TIME_OF_DAY ;	//compare time module 2
   dsv_info_mod_2 : WORD ;	//dataset info module 2
   data_0_mod_2 : WORD ;	//data 0 - 1 module 2
   data_2_mod_2 : WORD ;	//data 2 - 3 module 2
   data_4_mod_2 : WORD ;	//data 4 - 5 module 2
   data_6_mod_2 : WORD ;	//data 6 - 7 module 2
   data_8_mod_2 : WORD ;	//data 8 - 9 module 2
   data_10_mod_2 : WORD ;	//data 10 - 11 module 2
   data_12_mod_2 : WORD ;	//data 12 - 13 module 2
   data_14_mod_2 : WORD ;	//data 14 - 15 module 2
   data_16_mod_2 : WORD ;	//data 16 - 17 module 2
   data_18_mod_2 : WORD ;	//data 18 - 19 module 2
   data_20_mod_2 : WORD ;	//data 20 - 21 module 2
   data_22_mod_2 : WORD ;	//data 22 - 23 module 2
   data_24_mod_2 : WORD ;	//data 24 - 25 module 2
   data_26_mod_2 : WORD ;	//data 26 - 27 module 2
   data_28_mod_2 : WORD ;	//data 28 - 29 module 2
   data_30_mod_2 : WORD ;	//data 30 - 31 module 2
   data_32_mod_2 : WORD ;	//data 32 - 33 module 2
   data_34_mod_2 : WORD ;	//data 34 - 35 module 2
   data_36_mod_2 : WORD ;	//data 36 - 37 module 2
   data_38_mod_2 : WORD ;	//data 38 - 39 module 2
   spare_350 : WORD ;
   spare_352 : WORD ;
   spare_354 : WORD ;
   spare_356 : WORD ;
   spare_358 : WORD ;
   error_Com_2 : WORD ;	//error indication  Com  module 2
   error_nb_Com_2 : WORD ;	//error number indication  Com  module 2
   state_SFB52a_2 : WORD ;	//state SFB52 part 1 module 2
   state_SFB52b_2 : WORD ;	//state SFB52 part 2 module 2
   state_SFB53a_2 : WORD ;	//state SFB53 part 1 module 2
   state_SFB53b_2 : WORD ;	//state SFB53 part 2 module 2
   spare_372 : WORD ;
   error_date_mod_2 : DATE ;	//error date module 2
   error_time_mod_2 : TIME_OF_DAY ;	//error time module 2
   error_info_mod_2 : WORD ;	//error info read values module 2
   error_F_Module_mod_2 : WORD ;	//error safety module module 2
   error_F_DI_1_mod_2 : WORD ;	//error safety input 1 module 2
   error_F_DI_2_mod_2 : WORD ;	//error safety input 2 module 2
   error_F_DI_3_mod_2 : WORD ;	//error safety input 3 module 2
   error_F_DI_4_mod_2 : WORD ;	//error safety input 4 module 2
   error_F_DI_5_mod_2 : WORD ;	//error safety input 5 module 2
   error_F_DI_6_mod_2 : WORD ;	//error safety input 6 module 2
   error_F_DI_7_mod_2 : WORD ;	//error safety input 7 module 2
   error_F_DI_8_mod_2 : WORD ;	//error safety input 8 module 2
   error_F_DO_1_mod_2 : WORD ;	//error safety output 1 module 2
   error_F_DO_2_mod_2 : WORD ;	//error safety output 2 module 2
   error_F_DO_3_mod_2 : WORD ;	//error safety output 3 module 2
   error_F_DO_4_mod_2 : WORD ;	//error safety output 4 module 2
   error_Reg52_mod_2 : WORD ;	//error safety module register 52 module 2
   error_Reg53_mod_2 : WORD ;	//error safety module register 53 module 2
   error_Reg54_mod_2 : WORD ;	//error safety module register 54 module 2
   error_Reg55_mod_2 : WORD ;	//error safety module register 55 module 2
   spare_416 : WORD ;
   spare_418 : WORD ;
   comCountStart_3 : WORD ;	//comCountStart indication 3
   mod_type_3 : WORD ;	//module type 3
   mod_version_3 : WORD ;	//module version 3
   spare_426 : WORD ;
   spare_428 : WORD ;
   upl_date_mod_3 : DATE ;	//upload date module 3
   upl_time_mod_3 : TIME_OF_DAY ;	//upload time module 3
   dnl_date_mod_3 : DATE ;	//download date module 3
   dnl_time_mod_3 : TIME_OF_DAY ;	//download time module 3
   cmp_date_mod_3 : DATE ;	//compare date module  3
   cmp_time_mod_3 : TIME_OF_DAY ;	//compare time module  3
   dsv_info_mod_3 : WORD ;	//dataset info module 3
   data_0_mod_3 : WORD ;	//data 0 - 1 module 3
   data_2_mod_3 : WORD ;	//data 2 - 3 module 3
   data_4_mod_3 : WORD ;	//data 4 - 5 module 3
   data_6_mod_3 : WORD ;	//data 6 - 7 module 3
   data_8_mod_3 : WORD ;	//data 8 - 9 module 3
   data_10_mod_3 : WORD ;	//data 10 - 11 module 3
   data_12_mod_3 : WORD ;	//data 12 - 13 module 3
   data_14_mod_3 : WORD ;	//data 14 - 15 module 3
   data_16_mod_3 : WORD ;	//data 16 - 17 module 3
   data_18_mod_3 : WORD ;	//data 18 - 19 module 3
   data_20_mod_3 : WORD ;	//data 20 - 21 module 3
   data_22_mod_3 : WORD ;	//data 22 - 23 module 3
   data_24_mod_3 : WORD ;	//data 24 - 25 module 3
   data_26_mod_3 : WORD ;	//data 26 - 27 module 3
   data_28_mod_3 : WORD ;	//data 28 - 29 module 3
   data_30_mod_3 : WORD ;	//data 30 - 31 module 3
   data_32_mod_3 : WORD ;	//data 32 - 33 module 3
   data_34_mod_3 : WORD ;	//data 34 - 35 module 3
   data_36_mod_3 : WORD ;	//data 36 - 37 module 3
   data_38_mod_3 : WORD ;	//data 38 - 39 module 3
   spare_490 : WORD ;
   spare_492 : WORD ;
   spare_494 : WORD ;
   spare_496 : WORD ;
   spare_498 : WORD ;
   error_Com_3 : WORD ;	//error indication  Com  module 3
   error_nb_Com_3 : WORD ;	//error number indication  Com  module 3
   state_SFB52a_3 : WORD ;	//state SFB52 part 1 module 3
   state_SFB52b_3 : WORD ;	//state SFB52 part 2 module 3
   state_SFB53a_3 : WORD ;	//state SFB53 part 1 module 3
   state_SFB53b_3 : WORD ;	//state SFB53 part 2 module 3
   spare_512 : WORD ;
   error_date_mod_3 : DATE ;	//error date module 3
   error_time_mod_3 : TIME_OF_DAY ;	//error time module 3
   error_info_mod_3 : WORD ;	//error info read values module 3
   error_F_Module_mod_3 : WORD ;	//error safety module module 3
   error_F_DI_1_mod_3 : WORD ;	//error safety input 1 module 3
   error_F_DI_2_mod_3 : WORD ;	//error safety input 2 module 3
   error_F_DI_3_mod_3 : WORD ;	//error safety input 3 module 3
   error_F_DI_4_mod_3 : WORD ;	//error safety input 4 module 3
   error_F_DI_5_mod_3 : WORD ;	//error safety input 5 module 3
   error_F_DI_6_mod_3 : WORD ;	//error safety input 6 module 3
   error_F_DI_7_mod_3 : WORD ;	//error safety input 7 module 3
   error_F_DI_8_mod_3 : WORD ;	//error safety input 8 module 3
   error_F_DO_1_mod_3 : WORD ;	//error safety output 1 module 3
   error_F_DO_2_mod_3 : WORD ;	//error safety output 2 module 3
   error_F_DO_3_mod_3 : WORD ;	//error safety output 3 module 3
   error_F_DO_4_mod_3 : WORD ;	//error safety output 4 module 3
   error_Reg52_mod_3 : WORD ;	//error safety module register 52 module 3
   error_Reg53_mod_3 : WORD ;	//error safety module register 53 module 3
   error_Reg54_mod_3 : WORD ;	//error safety module register 54 module 3
   error_Reg55_mod_3 : WORD ;	//error safety module register 55 module 3
   spare_556 : WORD ;
   spare_558 : WORD ;
   comCountStart_4 : WORD ;	//comCountStart indication 4
   mod_type_4 : WORD ;	//module type  4
   mod_version_4 : WORD ;	//module version  4
   spare_566 : WORD ;
   spare_568 : WORD ;
   upl_date_mod_4 : DATE ;	//upload date module  4
   upl_time_mod_4 : TIME_OF_DAY ;	//upload time module  4
   dnl_date_mod_4 : DATE ;	//download date module  4
   dnl_time_mod_4 : TIME_OF_DAY ;	//download time module  4
   cmp_date_mod_4 : DATE ;	//compare date module   4
   cmp_time_mod_4 : TIME_OF_DAY ;	//compare time module   4
   dsv_info_mod_4 : WORD ;	//dataset info module 4
   data_0_mod_4 : WORD ;	//data 0 - 1 module  4
   data_2_mod_4 : WORD ;	//data 2 - 3 module  4
   data_4_mod_4 : WORD ;	//data 4 - 5 module  4
   data_6_mod_4 : WORD ;	//data 6 - 7 module  4
   data_8_mod_4 : WORD ;	//data 8 - 9 module  4
   data_10_mod_4 : WORD ;	//data 10 - 11 module  4
   data_12_mod_4 : WORD ;	//data 12 - 13 module  4
   data_14_mod_4 : WORD ;	//data 14 - 15 module  4
   data_16_mod_4 : WORD ;	//data 16 - 17 module  4
   data_18_mod_4 : WORD ;	//data 18 - 19 module  4
   data_20_mod_4 : WORD ;	//data 20 - 21 module  4
   data_22_mod_4 : WORD ;	//data 22 - 23 module  4
   data_24_mod_4 : WORD ;	//data 24 - 25 module  4
   data_26_mod_4 : WORD ;	//data 26 - 27 module  4
   data_28_mod_4 : WORD ;	//data 28 - 29 module  4
   data_30_mod_4 : WORD ;	//data 30 - 31 module  4
   data_32_mod_4 : WORD ;	//data 32 - 33 module  4
   data_34_mod_4 : WORD ;	//data 34 - 35 module  4
   data_36_mod_4 : WORD ;	//data 36 - 37 module  4
   data_38_mod_4 : WORD ;	//data 38 - 39 module  4
   spare_630 : WORD ;
   spare_632 : WORD ;
   spare_634 : WORD ;
   spare_636 : WORD ;
   spare_638 : WORD ;
   error_Com_4 : WORD ;	//error indication  Com  module 4
   error_nb_Com_4 : WORD ;	//error number indication  Com  module 4
   state_SFB52a_4 : WORD ;	//state SFB52 part 1 module 4
   state_SFB52b_4 : WORD ;	//state SFB52 part 2 module 4
   state_SFB53a_4 : WORD ;	//state SFB53 part 1 module 4
   state_SFB53b_4 : WORD ;	//state SFB53 part 2 module 4
   spare_652 : WORD ;
   error_date_mod_4 : DATE ;	//error date module 4
   error_time_mod_4 : TIME_OF_DAY ;	//error time module 4
   error_info_mod_4 : WORD ;	//error info read values module 4
   error_F_Module_mod_4 : WORD ;	//error safety module module 4
   error_F_DI_1_mod_4 : WORD ;	//error safety input 1 module 4
   error_F_DI_2_mod_4 : WORD ;	//error safety input 2 module 4
   error_F_DI_3_mod_4 : WORD ;	//error safety input 3 module 4
   error_F_DI_4_mod_4 : WORD ;	//error safety input 4 module 4
   error_F_DI_5_mod_4 : WORD ;	//error safety input 5 module 4
   error_F_DI_6_mod_4 : WORD ;	//error safety input 6 module 4
   error_F_DI_7_mod_4 : WORD ;	//error safety input 7 module 4
   error_F_DI_8_mod_4 : WORD ;	//error safety input 8 module 4
   error_F_DO_1_mod_4 : WORD ;	//error safety output 1 module 4
   error_F_DO_2_mod_4 : WORD ;	//error safety output 2 module 4
   error_F_DO_3_mod_4 : WORD ;	//error safety output 3 module 4
   error_F_DO_4_mod_4 : WORD ;	//error safety output 4 module 4
   error_Reg52_mod_4 : WORD ;	//error safety module register 52 module 4
   error_Reg53_mod_4 : WORD ;	//error safety module register 53 module 4
   error_Reg54_mod_4 : WORD ;	//error safety module register 54 module 4
   error_Reg55_mod_4 : WORD ;	//error safety module register 55 module 4
   spare_696 : WORD ;
   spare_698 : WORD ;
  END_STRUCT ;	
BEGIN
   versionInfo_1 := 37;
   versionInfo_2 := W#16#501;
   chkInfoData := W#16#1;
   fctReqTimeout := 6000;
   maxModules := 1;
   type_module_1 := 667;
   adr_module_1 := 55;
   bussystem_mod_1 := 1;
   bussystem_mod_2 := 1;
   bussystem_mod_3 := 1;
   bussystem_mod_4 := 1;
   slaveConfigInfo := DW#16#1;
   init_fb_done := DW#16#7;
   check_cfg_done := DW#16#6;
   upload_done := DW#16#7;
   download_done := DW#16#7;
   compare_done := DW#16#7;
   cmdCtrl_FB37 := W#16#FE00;
   comCountStart_1 := W#16#2;
   mod_type_1 := W#16#1A17;
   mod_version_1 := W#16#3;
   dsv_info_mod_1 := W#16#317C;
   data_0_mod_1 := W#16#4545;
   data_2_mod_1 := W#16#10CC;
   data_4_mod_1 := W#16#20CC;
   data_6_mod_1 := W#16#203;
   data_8_mod_1 := W#16#F430;
   data_10_mod_1 := W#16#6400;
   data_12_mod_1 := W#16#6400;
   data_18_mod_1 := W#16#3333;
   data_20_mod_1 := W#16#7C31;
   data_22_mod_1 := W#16#FEFF;
   data_24_mod_1 := W#16#9F5;
   data_26_mod_1 := W#16#3D5B;
   data_30_mod_1 := W#16#1E04;
   comCountStart_2 := W#16#2;
   mod_type_2 := W#16#1A17;
   mod_version_2 := W#16#3;
   dsv_info_mod_2 := W#16#7573;
   data_0_mod_2 := W#16#4545;
   data_2_mod_2 := W#16#10CC;
   data_4_mod_2 := W#16#20CC;
   data_6_mod_2 := W#16#203;
   data_8_mod_2 := W#16#F430;
   data_10_mod_2 := W#16#6400;
   data_12_mod_2 := W#16#6400;
   data_16_mod_2 := W#16#100;
   data_18_mod_2 := W#16#3733;
   data_20_mod_2 := W#16#7375;
   data_22_mod_2 := W#16#FEFF;
   data_24_mod_2 := W#16#B6E;
   data_26_mod_2 := W#16#5B54;
   data_30_mod_2 := W#16#7E16;
   comCountStart_3 := W#16#2;
   mod_type_3 := W#16#1A0D;
   mod_version_3 := W#16#3;
   dsv_info_mod_3 := W#16#B395;
   data_0_mod_3 := W#16#4545;
   data_2_mod_3 := W#16#10CC;
   data_4_mod_3 := W#16#20CC;
   data_6_mod_3 := W#16#204;
   data_8_mod_3 := W#16#F430;
   data_10_mod_3 := W#16#6400;
   data_12_mod_3 := W#16#6400;
   data_18_mod_3 := W#16#AA00;
   data_20_mod_3 := W#16#95B3;
   data_22_mod_3 := W#16#FEFF;
   data_24_mod_3 := W#16#CC3D;
   data_26_mod_3 := W#16#1256;
   data_30_mod_3 := W#16#E0D;
END_DATA_BLOCK

ORGANIZATION_BLOCK "CYCL_EXC"	// OB 1
TITLE = "Main Program Sweep (Cycle)"
VERSION : 0.1
VAR_TEMP
  OB1_EV_CLASS : BYTE ;	//Bits 0-3 = 1 (Coming event), Bits 4-7 = 1 (Event class 1)
  OB1_SCAN_1 : BYTE ;	//1 (Cold restart scan 1 of OB 1), 3 (Scan 2-n of OB 1)
  OB1_PRIORITY : BYTE ;	//Priority of OB Execution
  OB1_OB_NUMBR : BYTE ;	//1 (Organization block 1, OB1)
  OB1_RESERVED_1 : BYTE ;	//Reserved for system
  OB1_RESERVED_2 : BYTE ;	//Reserved for system
  OB1_PREV_CYCLE : INT ;	//Cycle time of previous OB1 scan (milliseconds)
  OB1_MIN_CYCLE : INT ;	//Minimum cycle time of OB1 (milliseconds)
  OB1_MAX_CYCLE : INT ;	//Maximum cycle time of OB1 (milliseconds)
  OB1_DATE_TIME : DATE_AND_TIME ;	//Date and time OB1 started
END_VAR
BEGIN
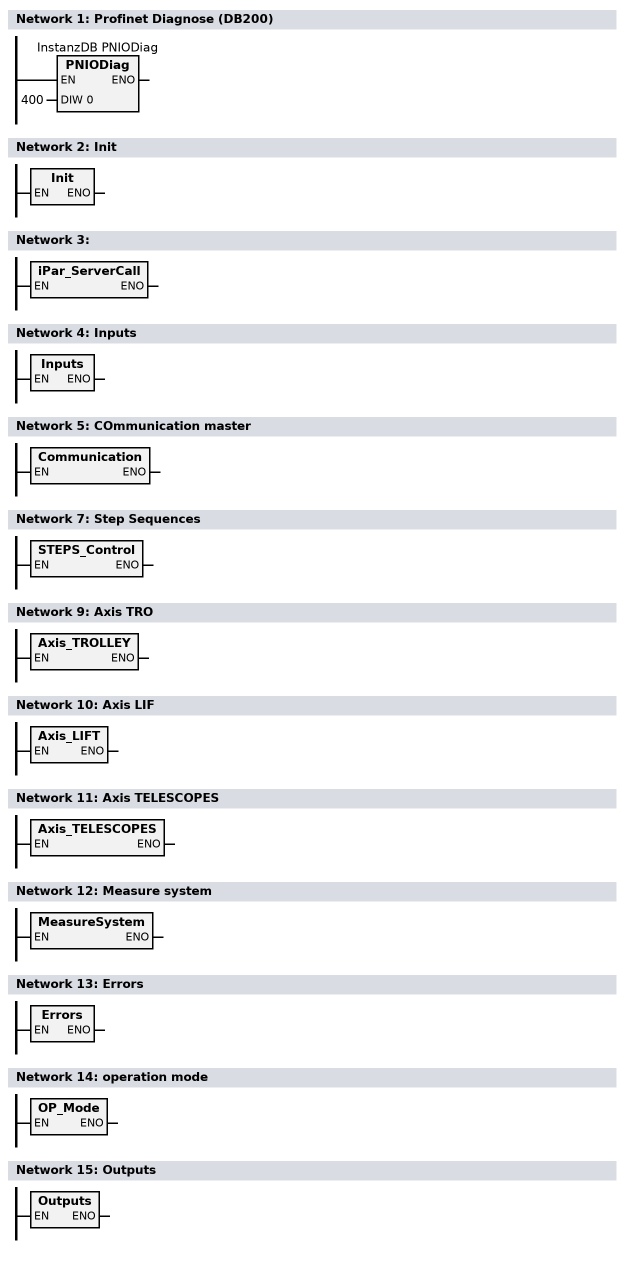
NETWORK
TITLE = Profinet Diagnose (DB200)
      CALL  "PNIODiag" , "InstanzDB PNIODiag" (
           DIW 0                    := 400);
      NOP   0;
NETWORK
TITLE = Init
      CALL  "Init";
      NOP   0;
NETWORK
TITLE =
      CALL  "iPar_ServerCall";
      NOP   0;
NETWORK
TITLE = Inputs
      CALL  "Inputs";
      NOP   0;
NETWORK
TITLE = COmmunication master
      CALL  "Communication";
      NOP   0;
NETWORK
TITLE = Main Cabinet
NETWORK
TITLE = Step Sequences
      CALL  "STEPS_Control";
      NOP   0;
NETWORK
TITLE = Axis BRI
NETWORK
TITLE = Axis TRO
      CALL  "Axis_TROLLEY";
      NOP   0;
NETWORK
TITLE = Axis LIF
      CALL  "Axis_LIFT";
      NOP   0;
NETWORK
TITLE = Axis TELESCOPES
      CALL  "Axis_TELESCOPES";
      NOP   0;
NETWORK
TITLE = Measure system
      CALL  "MeasureSystem";
      NOP   0;
NETWORK
TITLE = Errors
      CALL  "Errors";
      NOP   0;
NETWORK
TITLE = operation mode
      CALL  "OP_Mode";
      NOP   0;
NETWORK
TITLE = Outputs
      CALL  "Outputs";
      NOP   0;
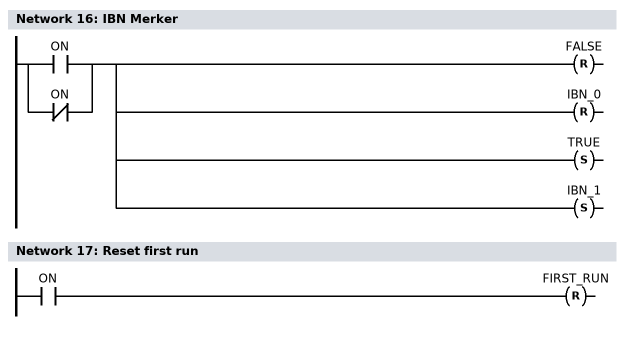
NETWORK
TITLE = IBN Merker
      O     "ON";
      ON    "ON";
      R     "FALSE";
      R     "IBN_0";
      S     "TRUE";
      S     "IBN_1";
NETWORK
TITLE = Reset first run
      A     "ON";
      R     "FIRST_RUN";
END_ORGANIZATION_BLOCK

ORGANIZATION_BLOCK "CYC_INT5"	// OB 35
TITLE = "Cyclic Interrupt"
VERSION : 0.1
VAR_TEMP
  OB35_EV_CLASS : BYTE ;	//Bits 0-3 = 1 (Coming event), Bits 4-7 = 1 (Event class 1)
  OB35_STRT_INF : BYTE ;	//16#36 (OB 35 has started)
  OB35_PRIORITY : BYTE ;	//Priority of OB Execution
  OB35_OB_NUMBR : BYTE ;	//35 (Organization block 35, OB35)
  OB35_RESERVED_1 : BYTE ;	//Reserved for system
  OB35_RESERVED_2 : BYTE ;	//Reserved for system
  OB35_PHASE_OFFSET : WORD ;	//Phase offset (msec)
  OB35_RESERVED_3 : INT ;	//Reserved for system
  OB35_EXC_FREQ : INT ;	//Frequency of execution (msec)
  OB35_DATE_TIME : DATE_AND_TIME ;	//Date and time OB35 started
END_VAR
BEGIN
NETWORK
TITLE =
      CALL  "F-CALL";
END_ORGANIZATION_BLOCK

ORGANIZATION_BLOCK "CYCL_FLT"	// OB 80
TITLE = "Cycle Time Fault"
VERSION : 0.1
VAR_TEMP
  OB80_EV_CLASS : BYTE ;	//16#35, Event class 3, Entering event state, Internal fault event
  OB80_FLT_ID : BYTE ;	//16#XX, Fault identifcation code
  OB80_PRIORITY : BYTE ;	//Priority of OB Execution
  OB80_OB_NUMBR : BYTE ;	//80 (Organization block 80, OB80)
  OB80_RESERVED_1 : BYTE ;	//Reserved for system
  OB80_RESERVED_2 : BYTE ;	//Reserved for system
  OB80_ERROR_INFO : WORD ;	//Error information on event
  OB80_ERR_EV_CLASS : BYTE ;	//Class of event causing error
  OB80_ERR_EV_NUM : BYTE ;	//Number of event causing error
  OB80_OB_PRIORITY : BYTE ;	//Priority of OB causing error
  OB80_OB_NUM : BYTE ;	//Number of OB causing error
  OB80_DATE_TIME : DATE_AND_TIME ;	//Date and time OB80 started
END_VAR
BEGIN
// (block stored without names or comments; labels and parameter names are numbered)
END_ORGANIZATION_BLOCK

ORGANIZATION_BLOCK "I/O_FLT1"	// OB 82
TITLE = "I/O Point Fault"
AUTHOR : Koenig
VERSION : 0.1
VAR_TEMP
  OB82_EV_CLASS : BYTE ;	//16#39, Event class 3, Entering event state, Internal fault event
  OB82_FLT_ID : BYTE ;	//16#XX, Fault identifcation code
  OB82_PRIORITY : BYTE ;	//Priority of OB Execution
  OB82_OB_NUMBR : BYTE ;	//82 (Organization block 82, OB82)
  OB82_RESERVED_1 : BYTE ;	//Reserved for system
  OB82_IO_FLAG : BYTE ;	//Input (01010100), Output (01010101)
  OB82_MDL_ADDR : WORD ;	//Base address of module with fault
  OB82_MDL_DEFECT : BOOL ;	//Module defective
  OB82_INT_FAULT : BOOL ;	//Internal fault
  OB82_EXT_FAULT : BOOL ;	//External fault
  OB82_PNT_INFO : BOOL ;	//Point information
  OB82_EXT_VOLTAGE : BOOL ;	//External voltage low
  OB82_FLD_CONNCTR : BOOL ;	//Field wiring connector missing
  OB82_NO_CONFIG : BOOL ;	//Module has no configuration data
  OB82_CONFIG_ERR : BOOL ;	//Module has configuration error
  OB82_MDL_TYPE : BYTE ;	//Type of module
  OB82_SUB_MDL_ERR : BOOL ;	//Sub-Module is missing or has error
  OB82_COMM_FAULT : BOOL ;	//Communication fault
  OB82_MDL_STOP : BOOL ;	//Module is stopped
  OB82_WTCH_DOG_FLT : BOOL ;	//Watch dog timer stopped module
  OB82_INT_PS_FLT : BOOL ;	//Internal power supply fault
  OB82_PRIM_BATT_FLT : BOOL ;	//Primary battery is in fault
  OB82_BCKUP_BATT_FLT : BOOL ;	//Backup battery is in fault
  OB82_RESERVED_2 : BOOL ;	//Reserved for system
  OB82_RACK_FLT : BOOL ;	//Rack fault, only for bus interface module
  OB82_PROC_FLT : BOOL ;	//Processor fault
  OB82_EPROM_FLT : BOOL ;	//EPROM fault
  OB82_RAM_FLT : BOOL ;	//RAM fault
  OB82_ADU_FLT : BOOL ;	//ADU fault
  OB82_FUSE_FLT : BOOL ;	//Fuse fault
  OB82_HW_INTR_FLT : BOOL ;	//Hardware interupt input in fault
  OB82_RESERVED_3 : BOOL ;	//Reserved for system
  OB82_DATE_TIME : DATE_AND_TIME ;	//Date and time OB82 started
END_VAR
BEGIN
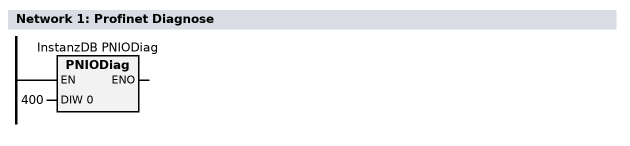
NETWORK
TITLE = Profinet Diagnose
      CALL  "PNIODiag" , "InstanzDB PNIODiag" (
           DIW 0                    := 400);
      NOP   0;
END_ORGANIZATION_BLOCK

ORGANIZATION_BLOCK "I/O_FLT2"	// OB 83
TITLE = "I/O Point Fault"
AUTHOR : Koenig
VERSION : 0.1
VAR_TEMP
  OB83_EV_CLASS : BYTE ;	//16#38/39, Event class 3, module inserted/removed (8/9)
  OB83_FLT_ID : BYTE ;	//16#XX, Fault identifcation code
  OB83_PRIORITY : BYTE ;	//Priority of OB Execution
  OB83_OB_NUMBR : BYTE ;	//83 (Organization block 83, OB83)
  OB83_RESERVED_1 : BYTE ;	//Reserved for system
  OB83_MDL_ID : BYTE ;	//Input module (01010100), Output module (01010101)
  OB83_MDL_ADDR : WORD ;	//Base address of module with point fault
  OB83_RACK_NUM : INT ;	//Number of rack that has module with point fault
  OB83_MDL_TYPE : WORD ;	//Module type with point fault
  OB83_DATE_TIME : DATE_AND_TIME ;	//Date and time OB83 started
END_VAR
BEGIN
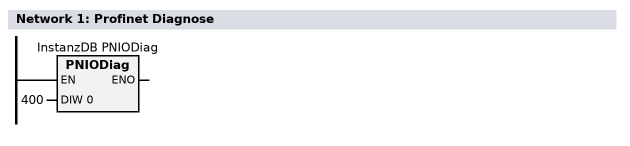
NETWORK
TITLE = Profinet Diagnose
      CALL  "PNIODiag" , "InstanzDB PNIODiag" (
           DIW 0                    := 400);
      NOP   0;
END_ORGANIZATION_BLOCK

ORGANIZATION_BLOCK "OBNL_FLT"	// OB 85
TITLE = "Organization Block (OB) Not Loaded Fault"
AUTHOR : Koenig
VERSION : 0.1
VAR_TEMP
  OB85_EV_CLASS : BYTE ;	//16#35 Event class 3
  OB85_FLT_ID : BYTE ;	//16#XX, Fault identification code
  OB85_PRIORITY : BYTE ;	//Priority of OB Execution
  OB85_OB_NUMBR : BYTE ;	//85 (Organization block 85, OB85)
  OB85_RESERVED_1 : BYTE ;	//Reserved for system
  OB85_RESERVED_2 : BYTE ;	//Reserved for system
  OB85_RESERVED_3 : INT ;	//Reserved for system
  OB85_ERR_EV_CLASS : BYTE ;	//Class of event causing error
  OB85_ERR_EV_NUM : BYTE ;	//Number of event causing error
  OB85_OB_PRIOR : BYTE ;	//Priority of OB causing error
  OB85_OB_NUM : BYTE ;	//Number of OB causing error
  OB85_DATE_TIME : DATE_AND_TIME ;	//Date and time OB85 started
END_VAR
BEGIN
NETWORK
TITLE =
END_ORGANIZATION_BLOCK

ORGANIZATION_BLOCK "RACK_FLT"	// OB 86
TITLE = "Loss Of Rack Fault"
AUTHOR : Koenig
VERSION : 0.1
VAR_TEMP
  OB86_EV_CLASS : BYTE ;	//16#38/39 Event class 3
  OB86_FLT_ID : BYTE ;	//16#C1/C4/C5, Fault identifcation code
  OB86_PRIORITY : BYTE ;	//Priority of OB Execution
  OB86_OB_NUMBR : BYTE ;	//86 (Organization block 86, OB86)
  OB86_RESERVED_1 : BYTE ;	//Reserved for system
  OB86_RESERVED_2 : BYTE ;	//Reserved for system
  OB86_MDL_ADDR : WORD ;	//Base address of IM module in rack with fault
  OB86_RACKS_FLTD : ARRAY  [0 .. 31 ] OF BOOL ;	//Racks in fault
  OB86_DATE_TIME : DATE_AND_TIME ;	//Date and time OB86 started
END_VAR
BEGIN
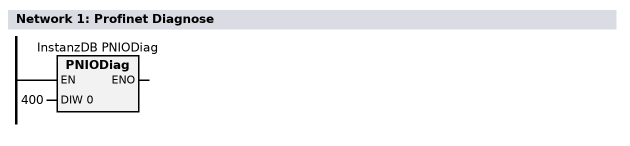
NETWORK
TITLE = Profinet Diagnose
      CALL  "PNIODiag" , "InstanzDB PNIODiag" (
           DIW 0                    := 400);
      NOP   0;
END_ORGANIZATION_BLOCK

ORGANIZATION_BLOCK "COMM_FLT"	// OB 87
TITLE = "Communication Fault"
AUTHOR : Koenig
VERSION : 0.1
VAR_TEMP
  OB87_EV_CLASS : BYTE ;	//16#39 Event class 3
  OB87_FLT_ID : BYTE ;	//16#XX, Fault identifcation code
  OB87_PRIORITY : BYTE ;	//Priority of OB Execution
  OB87_OB_NUMBR : BYTE ;	//87 (Organization block 87, OB87)
  OB87_RESERVED_1 : BYTE ;	//Reserved for system
  OB87_RESERVED_2 : BYTE ;	//Reserved for system
  OB87_RESERVED_3 : WORD ;	//Reserved for system
  OB87_RESERVED_4 : DWORD ;	//Reserved for system
  OB87_DATE_TIME : DATE_AND_TIME ;	//Date and time OB87 started
END_VAR
BEGIN
NETWORK
TITLE =
END_ORGANIZATION_BLOCK

ORGANIZATION_BLOCK "STARTUP"	// OB 100
TITLE = "Complete Restart"
AUTHOR : Koenig
VERSION : 0.1
VAR_TEMP
  OB100_EV_CLASS : BYTE ;	//16#13, Event class 1, Entering event state, Event logged in diagnostic buffer
  OB100_STRTUP : BYTE ;	//16#81/82/83/84 Method of startup
  OB100_PRIORITY : BYTE ;	//Priority of OB Execution
  OB100_OB_NUMBR : BYTE ;	//100 (Organization block 100, OB100)
  OB100_RESERVED_1 : BYTE ;	//Reserved for system
  OB100_RESERVED_2 : BYTE ;	//Reserved for system
  OB100_STOP : WORD ;	//Event that caused CPU to stop (16#4xxx)
  OB100_STRT_INFO : DWORD ;	//Information on how system started
  OB100_DATE_TIME : DATE_AND_TIME ;	//Date and time OB100 started
  ZeroDouble : DINT ;
  ret : INT ;
END_VAR
BEGIN
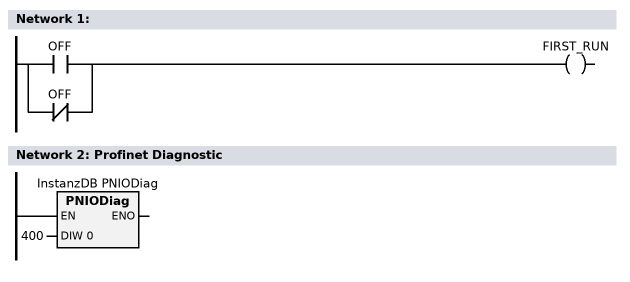
NETWORK
TITLE =
      O     "OFF";
      ON    "OFF";
      =     "FIRST_RUN";
NETWORK
TITLE = Profinet Diagnostic
      CALL  "PNIODiag" , "InstanzDB PNIODiag" (
           DIW 0                    := 400);
      NOP   0;
END_ORGANIZATION_BLOCK

ORGANIZATION_BLOCK "PROG_ERR"	// OB 121
TITLE = "Programming Error"
AUTHOR : Koenig
VERSION : 0.1
VAR_TEMP
  OB121_EV_CLASS : BYTE ;	//16#25, Event class 2, Entering event state, Internal fault event
  OB121_SW_FLT : BYTE ;	//16#XX Software programming fault
  OB121_PRIORITY : BYTE ;	//Priority of OB Execution
  OB121_OB_NUMBR : BYTE ;	//121 (Organization block 121, OB121)
  OB121_BLK_TYPE : BYTE ;	//16#88/8A/8B/8C/8E Type of block fault occured in
  OB121_RESERVED_1 : BYTE ;	//Reserved for system
  OB121_FLT_REG : WORD ;	//16#XX Specific register that caused fault
  OB121_BLK_NUM : WORD ;	//Number of block that programming fault occured in
  OB121_PRG_ADDR : WORD ;	//Address in block where programming fault occured
  OB121_DATE_TIME : DATE_AND_TIME ;	//Date and time OB121 started
END_VAR
BEGIN
// (block stored without names or comments; labels and parameter names are numbered)
END_ORGANIZATION_BLOCK

ORGANIZATION_BLOCK "MOD_ERR"	// OB 122
TITLE = "Module Access Error"
AUTHOR : Koenig
VERSION : 0.1
VAR_TEMP
  OB122_EV_CLASS : BYTE ;	//16#29, Event class 2, Entering event state, Internal fault event
  OB122_SW_FLT : BYTE ;	//16#XX Software error code
  OB122_PRIORITY : BYTE ;	//Priority of OB Execution
  OB122_OB_NUMBR : BYTE ;	//122 (Organization block 122, OB122)
  OB122_BLK_TYPE : BYTE ;	//16#88/8C/8E Type of block fault occured in
  OB122_MEM_AREA : BYTE ;	//Memory area where access error occured
  OB122_MEM_ADDR : WORD ;	//Memory address where access error occured
  OB122_BLK_NUM : WORD ;	//Block number in which error occured
  OB122_PRG_ADDR : WORD ;	//Program address where error occured
  OB122_DATE_TIME : DATE_AND_TIME ;	//Date and time OB1 started
END_VAR
BEGIN
NETWORK
TITLE =
END_ORGANIZATION_BLOCK

SYMBOL_TABLE
"DBS_Input"	DB 100	DB 100
"DBS_Output"	DB 110	DB 110
"DB_Input"	DB 1000	DB 1000
"DB_Output"	DB 1010	DB 1010
"FCS_Input"	FC 100	FC 100
"FCS_Output"	FC 110	FC 110
"FC_Input"	FC 1000	FC 1000
"FC_Output"	FC 1010	FC 1010
"ES_020_0"	I 20.0	BOOL	// IN emergency stop extern CH1
"ES_020_1"	I 20.1	BOOL	// IN emergency stop extern CH2
"ES_020_2"	I 20.2	BOOL	// Spare
"ES_020_3"	I 20.3	BOOL	// Spare
"ES_025_0"	I 25.0	BOOL	// Emergency stop CH1
"ES_025_1"	I 25.1	BOOL	// Emergency stop CH2
"ES_025_2"	I 25.2	BOOL	// Spare
"ES_025_3"	I 25.3	BOOL	// Spare
"ES_025_4"	I 25.4	BOOL	// Automatic mode CH1
"ES_025_5"	I 25.5	BOOL	// Automatic mode CH2
"ES_025_6"	I 25.6	BOOL	// Service mode CH1
"ES_025_7"	I 25.7	BOOL	// Service mode CH2
"ES_050_0"	I 50.0	BOOL	// Spare
"ES_050_1"	I 50.1	BOOL	// IN BRI fast stop
"ES_050_2"	I 50.2	BOOL	// IN LIF fast stop
"ES_050_3"	I 50.3	BOOL	// IN WID fast stop
"ES_055_0"	I 55.0	BOOL	// Spare
"ES_055_1"	I 55.1	BOOL	// IN emergency stop CH1/2
"ES_055_2"	I 55.2	BOOL	// LIF overland NC
"ES_055_3"	I 55.3	BOOL	// LIF slack cable NC
"ES_060_0"	I 60.0	BOOL	// WID left rocker switch on CH1
"ES_060_1"	I 60.1	BOOL	// WID left rocker switch on CH2
"ES_060_2"	I 60.2	BOOL	// WID left rocker switch off CH1
"ES_060_3"	I 60.3	BOOL	// WID left rocker switch off CH2
"ES_060_4"	I 60.4	BOOL	// WID left panel switch on CH1
"ES_060_5"	I 60.5	BOOL	// WID left panel switch on CH2
"ES_060_6"	I 60.6	BOOL	// WID left panel switch off CH1
"ES_060_7"	I 60.7	BOOL	// WID left panel switch off CH2
"ES_065_0"	I 65.0	BOOL	// WID right rocker switch on CH1
"ES_065_1"	I 65.1	BOOL	// WID right rocker switch on CH2
"ES_065_2"	I 65.2	BOOL	// WID right rocker switch off CH1
"ES_065_3"	I 65.3	BOOL	// WID right rocker switch off CH2
"ES_065_4"	I 65.4	BOOL	// WID right panel switch on CH1
"ES_065_5"	I 65.5	BOOL	// WID right panel switch on CH2
"ES_065_6"	I 65.6	BOOL	// WID right panel switch off CH1
"ES_065_7"	I 65.7	BOOL	// WID right panel switch off CH2
"ES_070_0"	I 70.0	BOOL	// Safety bar close CH1
"ES_070_1"	I 70.1	BOOL	// Safety bar close CH2
"ES_070_2"	I 70.2	BOOL	// Scanner 1 OSSD1
"ES_070_3"	I 70.3	BOOL	// Scanner 1 OSSD2
"ES_070_4"	I 70.4	BOOL	// Spare
"ES_070_5"	I 70.5	BOOL	// Spare
"ES_070_6"	I 70.6	BOOL	// Spare
"ES_070_7"	I 70.7	BOOL	// Spare
"ES_075_0"	I 75.0	BOOL	// Spare
"ES_075_1"	I 75.1	BOOL	// Spare
"ES_075_2"	I 75.2	BOOL	// Spare
"ES_075_3"	I 75.3	BOOL	// Spare
"ES_075_4"	I 75.4	BOOL	// No emergency stop
"ES_075_5"	I 75.5	BOOL	// No overtemp brake
"ES_075_6"	I 75.6	BOOL	// Bypass mode CH1
"ES_075_7"	I 75.7	BOOL	// Bypass mode CH2
"E100_0"	I 100.0	BOOL	// Spare
"E100_1"	I 100.1	BOOL	// Fuse 24V DC
"E100_2"	I 100.2	BOOL	// Overtemp cabinet
"E100_3"	I 100.3	BOOL	// Phase monitoring
"E100_4"	I 100.4	BOOL	// Spare
"E100_5"	I 100.5	BOOL	// Spare
"E100_6"	I 100.6	BOOL	// Spare
"E100_7"	I 100.7	BOOL	// Spare
"E101_0"	I 101.0	BOOL	// Button automatic
"E101_1"	I 101.1	BOOL	// Button reset
"E101_2"	I 101.2	BOOL	// Spare
"E101_3"	I 101.3	BOOL	// Spare
"E101_4"	I 101.4	BOOL	// Spare
"E101_5"	I 101.5	BOOL	// Button emergency stop 1
"E101_6"	I 101.6	BOOL	// Button emergency stop 2
"E101_7"	I 101.7	BOOL	// Button emergency stop 3
"E102_0"	I 102.0	BOOL	// Spare
"E102_1"	I 102.1	BOOL	// Spare
"E102_2"	I 102.2	BOOL	// Spare
"E102_3"	I 102.3	BOOL	// Spare
"E102_4"	I 102.4	BOOL	// Spare
"E102_5"	I 102.5	BOOL	// Spare
"E102_6"	I 102.6	BOOL	// Spare
"E102_7"	I 102.7	BOOL	// Spare
"E103_0"	I 103.0	BOOL	// Spare
"E103_1"	I 103.1	BOOL	// Spare
"E103_2"	I 103.2	BOOL	// Spare
"E103_3"	I 103.3	BOOL	// Spare
"E103_4"	I 103.4	BOOL	// Spare
"E103_5"	I 103.5	BOOL	// Spare
"E103_6"	I 103.6	BOOL	// Spare
"E103_7"	I 103.7	BOOL	// Spare
"E110_0"	I 110.0	BOOL	// Fuse cooling cabinet VEH
"E110_1"	I 110.1	BOOL	// Fuse 24V DC VEH
"E110_2"	I 110.2	BOOL	// Overtemp cabinet VEH
"E110_3"	I 110.3	BOOL	// Phase monitoring VEH
"E110_4"	I 110.4	BOOL	// Fuse 480V AC VEH
"E110_5"	I 110.5	BOOL	// Fuse brake
"E110_6"	I 110.6	BOOL	// Fuse safety bar
"E110_7"	I 110.7	BOOL	// Fan cabinet
"E111_0"	I 111.0	BOOL	// Spare
"E111_1"	I 111.1	BOOL	// Button reset VEH
"E111_2"	I 111.2	BOOL	// Spare
"E111_3"	I 111.3	BOOL	// Spare
"E111_4"	I 111.4	BOOL	// Scanner 1 error
"E111_5"	I 111.5	BOOL	// Scanner 1 warning
"E111_6"	I 111.6	BOOL	// Spare
"E111_7"	I 111.7	BOOL	// Spare
"E112_0"	I 112.0	BOOL	// BRI limit switch minus
"E112_1"	I 112.1	BOOL	// BRI limit switch plus
"E112_2"	I 112.2	BOOL	// LIF limit switch minus
"E112_3"	I 112.3	BOOL	// LIF limit switch plus
"E112_4"	I 112.4	BOOL	// LIF top NO
"E112_5"	I 112.5	BOOL	// LIF top NC
"E112_6"	I 112.6	BOOL	// Spare
"E112_7"	I 112.7	BOOL	// Spare
"E113_0"	I 113.0	BOOL	// LIF overload left
"E113_1"	I 113.1	BOOL	// LIF overload right
"E113_2"	I 113.2	BOOL	// LIF slack cable left
"E113_3"	I 113.3	BOOL	// LIF slack cable right
"E113_4"	I 113.4	BOOL	// Spare
"E113_5"	I 113.5	BOOL	// Spare
"E113_6"	I 113.6	BOOL	// Spare
"E113_7"	I 113.7	BOOL	// Spare
"E114_0"	I 114.0	BOOL	// Spare
"E114_1"	I 114.1	BOOL	// Spare
"E114_2"	I 114.2	BOOL	// WID left limit switch plus
"E114_3"	I 114.3	BOOL	// WID left limit switch minus
"E114_4"	I 114.4	BOOL	// WID right limit switch plus
"E114_5"	I 114.5	BOOL	// WID right limit switch minus
"E114_6"	I 114.6	BOOL	// WID left spike
"E114_7"	I 114.7	BOOL	// WID right spike
"E115_0"	I 115.0	BOOL	// Spare
"E115_1"	I 115.1	BOOL	// Spare
"E115_2"	I 115.2	BOOL	// Spare
"E115_3"	I 115.3	BOOL	// Spare
"E115_4"	I 115.4	BOOL	// Spare
"E115_5"	I 115.5	BOOL	// Spare
"E115_6"	I 115.6	BOOL	// Spare
"E115_7"	I 115.7	BOOL	// Spare
"E116_0"	I 116.0	BOOL	// IO storage free Q1
"E116_1"	I 116.1	BOOL	// IO storage free Q2
"E116_2"	I 116.2	BOOL	// Safety bar opened NO
"E116_3"	I 116.3	BOOL	// Safety bar opened NC
"E116_4"	I 116.4	BOOL	// Safety bar closed NO
"E116_5"	I 116.5	BOOL	// Safety bar closed NC
"E116_6"	I 116.6	BOOL	// Safety bar free left NO
"E116_7"	I 116.7	BOOL	// Safety bar free left NC
"E117_0"	I 117.0	BOOL	// Safety bar free right NO
"E117_1"	I 117.1	BOOL	// Saftey bar free right NC
"E117_2"	I 117.2	BOOL	// Spare
"E117_3"	I 117.3	BOOL	// Spare
"E117_4"	I 117.4	BOOL	// Spare
"E117_5"	I 117.5	BOOL	// Spare
"E117_6"	I 117.6	BOOL	// Spare
"E117_7"	I 117.7	BOOL	// Spare
"SYS_ON"	M 1.0	BOOL
"SYS_OFF"	M 1.1	BOOL
"SYS_TRUE"	M 1.2	BOOL
"SYS_FALSE"	M 1.3	BOOL
"IBN_ON"	M 100.0	BOOL
"IBN_OFF"	M 100.1	BOOL
"IBN_Test_1"	M 100.2	BOOL
"IBN_Test_2"	M 100.3	BOOL
"IBN_Test_3"	M 100.4	BOOL
"IBN_Test_4"	M 100.5	BOOL
"AS_020_0"	Q 20.0	BOOL	// OUT emergency stop extern CH1
"AS_020_1"	Q 20.1	BOOL	// OUT Emergency stop extern CH2
"AS_020_2"	Q 20.2	BOOL	// Spare
"AS_020_3"	Q 20.3	BOOL	// Spare
"AS_050_0"	Q 50.0	BOOL	// Spare
"AS_050_1"	Q 50.1	BOOL	// OUT BRI fast stop
"AS_050_2"	Q 50.2	BOOL	// OUT LIF fast stop
"AS_050_3"	Q 50.3	BOOL	// OUT WID fast stop
"AS_055_0"	Q 55.0	BOOL	// Spare
"AS_055_1"	Q 55.1	BOOL	// Spare
"AS_055_2"	Q 55.2	BOOL	// OUT emergency stop CH1
"AS_055_3"	Q 55.3	BOOL	// OUT emergency stop CH2
"A100_0"	Q 100.0	BOOL	// Spare
"A100_1"	Q 100.1	BOOL	// Fuse 24V DC reset
"A100_2"	Q 100.2	BOOL	// Spare
"A100_3"	Q 100.3	BOOL	// Spare
"A100_4"	Q 100.4	BOOL	// Spare
"A100_5"	Q 100.5	BOOL	// Status LED Bit0
"A100_6"	Q 100.6	BOOL	// Status LED Bit1
"A100_7"	Q 100.7	BOOL	// Status LED Bit2
"A101_0"	Q 101.0	BOOL	// LED automatic
"A101_1"	Q 101.1	BOOL	// LED reset
"A101_2"	Q 101.2	BOOL	// Spare
"A101_3"	Q 101.3	BOOL	// Spare
"A101_4"	Q 101.4	BOOL	// Spare
"A101_5"	Q 101.5	BOOL	// Spare
"A101_6"	Q 101.6	BOOL	// Spare
"A101_7"	Q 101.7	BOOL	// Spare
"A102_0"	Q 102.0	BOOL	// Emergency stop reset
"A102_1"	Q 102.1	BOOL	// Spare
"A102_2"	Q 102.2	BOOL	// Spare
"A102_3"	Q 102.3	BOOL	// Spare
"A102_4"	Q 102.4	BOOL	// Spare
"A102_5"	Q 102.5	BOOL	// Spare
"A102_6"	Q 102.6	BOOL	// Spare
"A102_7"	Q 102.7	BOOL	// Spare
"A110_0"	Q 110.0	BOOL	// Spare
"A110_1"	Q 110.1	BOOL	// Fuse 24V DC reset VEH
"A110_2"	Q 110.2	BOOL	// Spare
"A110_3"	Q 110.3	BOOL	// LED reset VEH
"A110_4"	Q 110.4	BOOL	// Sound generator
"A110_5"	Q 110.5	BOOL	// Status LED Bit0 VEH
"A110_6"	Q 110.6	BOOL	// Status LED Bit1 VEH
"A110_7"	Q 110.7	BOOL	// Status LED Bit2 VEH
"A111_0"	Q 111.0	BOOL	// Emergency stop reset VEH
"A111_1"	Q 111.1	BOOL	// Spare
"A111_2"	Q 111.2	BOOL	// Spare
"A111_3"	Q 111.3	BOOL	// Spare
"A111_4"	Q 111.4	BOOL	// Scanner on
"A111_5"	Q 111.5	BOOL	// Scanner field A
"A111_6"	Q 111.6	BOOL	// Scanner field B
"A111_7"	Q 111.7	BOOL	// Spare
"A112_0"	Q 112.0	BOOL	// Spare
"A112_1"	Q 112.1	BOOL	// Spare
"A112_2"	Q 112.2	BOOL	// Safety bar open
"A112_3"	Q 112.3	BOOL	// Safety bar close
"A112_4"	Q 112.4	BOOL	// Spare
"A112_5"	Q 112.5	BOOL	// Spare
"A112_6"	Q 112.6	BOOL	// Spare
"A112_7"	Q 112.7	BOOL	// Spare
END_SYMBOL_TABLE

FUNCTION "FCS_Input" : VOID	// FC 100
AUTHOR : Broecker
VERSION : 0.1
BEGIN
// body was compiled from another editor; compiled code not shown
END_FUNCTION

FUNCTION "FCS_Output" : VOID	// FC 110
AUTHOR : Broecker
VERSION : 0.1
BEGIN
// body was compiled from another editor; compiled code not shown
END_FUNCTION

FUNCTION "FC_Input" : VOID	// FC 1000
AUTHOR : Broecker
VERSION : 0.1
BEGIN
NETWORK
TITLE =
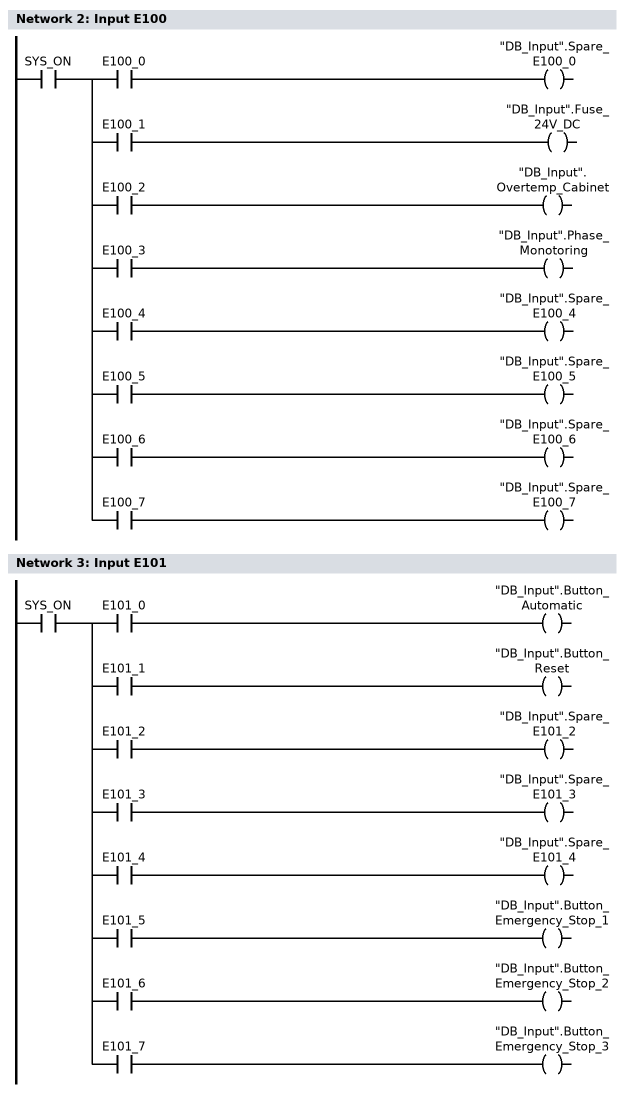
NETWORK
TITLE = Input E100
      A     "SYS_ON";
      =     L 0.0;
      A     L 0.0;
      A     "E100_0";
      =     "DB_Input".Spare_E100_0;
      A     L 0.0;
      A     "E100_1";
      =     "DB_Input".Fuse_24V_DC;
      A     L 0.0;
      A     "E100_2";
      =     "DB_Input".Overtemp_Cabinet;
      A     L 0.0;
      A     "E100_3";
      =     "DB_Input".Phase_Monotoring;
      A     L 0.0;
      A     "E100_4";
      =     "DB_Input".Spare_E100_4;
      A     L 0.0;
      A     "E100_5";
      =     "DB_Input".Spare_E100_5;
      A     L 0.0;
      A     "E100_6";
      =     "DB_Input".Spare_E100_6;
      A     L 0.0;
      A     "E100_7";
      =     "DB_Input".Spare_E100_7;
NETWORK
TITLE = Input E101
      A     "SYS_ON";
      =     L 0.0;
      A     L 0.0;
      A     "E101_0";
      =     "DB_Input".Button_Automatic;
      A     L 0.0;
      A     "E101_1";
      =     "DB_Input".Button_Reset;
      A     L 0.0;
      A     "E101_2";
      =     "DB_Input".Spare_E101_2;
      A     L 0.0;
      A     "E101_3";
      =     "DB_Input".Spare_E101_3;
      A     L 0.0;
      A     "E101_4";
      =     "DB_Input".Spare_E101_4;
      A     L 0.0;
      A     "E101_5";
      =     "DB_Input".Button_Emergency_Stop_1;
      A     L 0.0;
      A     "E101_6";
      =     "DB_Input".Button_Emergency_Stop_2;
      A     L 0.0;
      A     "E101_7";
      =     "DB_Input".Button_Emergency_Stop_3;
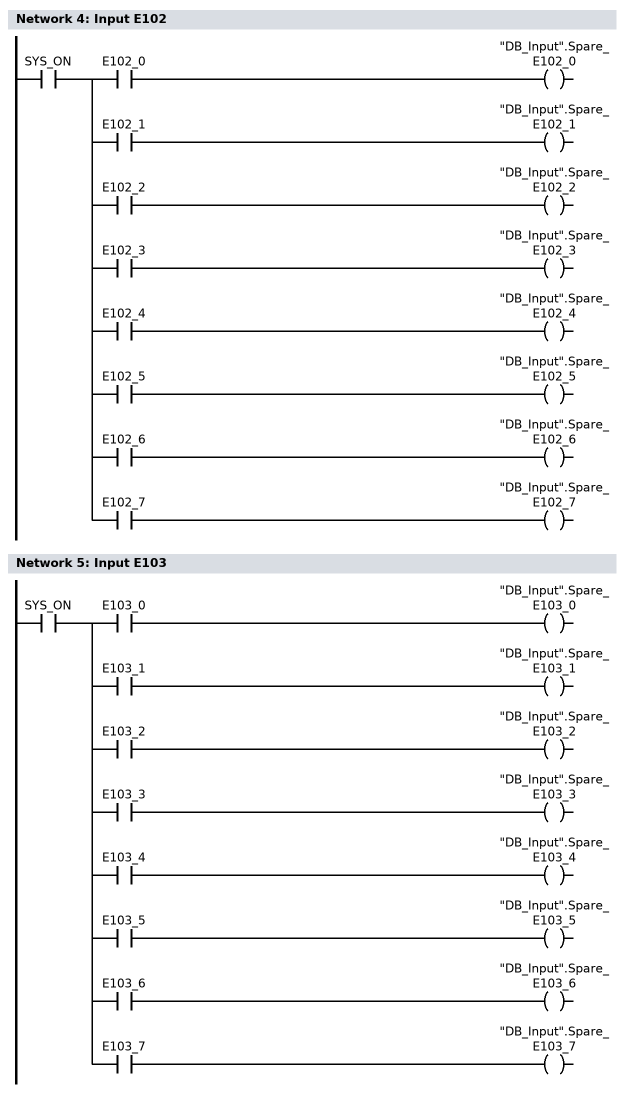
NETWORK
TITLE = Input E102
      A     "SYS_ON";
      =     L 0.0;
      A     L 0.0;
      A     "E102_0";
      =     "DB_Input".Spare_E102_0;
      A     L 0.0;
      A     "E102_1";
      =     "DB_Input".Spare_E102_1;
      A     L 0.0;
      A     "E102_2";
      =     "DB_Input".Spare_E102_2;
      A     L 0.0;
      A     "E102_3";
      =     "DB_Input".Spare_E102_3;
      A     L 0.0;
      A     "E102_4";
      =     "DB_Input".Spare_E102_4;
      A     L 0.0;
      A     "E102_5";
      =     "DB_Input".Spare_E102_5;
      A     L 0.0;
      A     "E102_6";
      =     "DB_Input".Spare_E102_6;
      A     L 0.0;
      A     "E102_7";
      =     "DB_Input".Spare_E102_7;
NETWORK
TITLE = Input E103
      A     "SYS_ON";
      =     L 0.0;
      A     L 0.0;
      A     "E103_0";
      =     "DB_Input".Spare_E103_0;
      A     L 0.0;
      A     "E103_1";
      =     "DB_Input".Spare_E103_1;
      A     L 0.0;
      A     "E103_2";
      =     "DB_Input".Spare_E103_2;
      A     L 0.0;
      A     "E103_3";
      =     "DB_Input".Spare_E103_3;
      A     L 0.0;
      A     "E103_4";
      =     "DB_Input".Spare_E103_4;
      A     L 0.0;
      A     "E103_5";
      =     "DB_Input".Spare_E103_5;
      A     L 0.0;
      A     "E103_6";
      =     "DB_Input".Spare_E103_6;
      A     L 0.0;
      A     "E103_7";
      =     "DB_Input".Spare_E103_7;
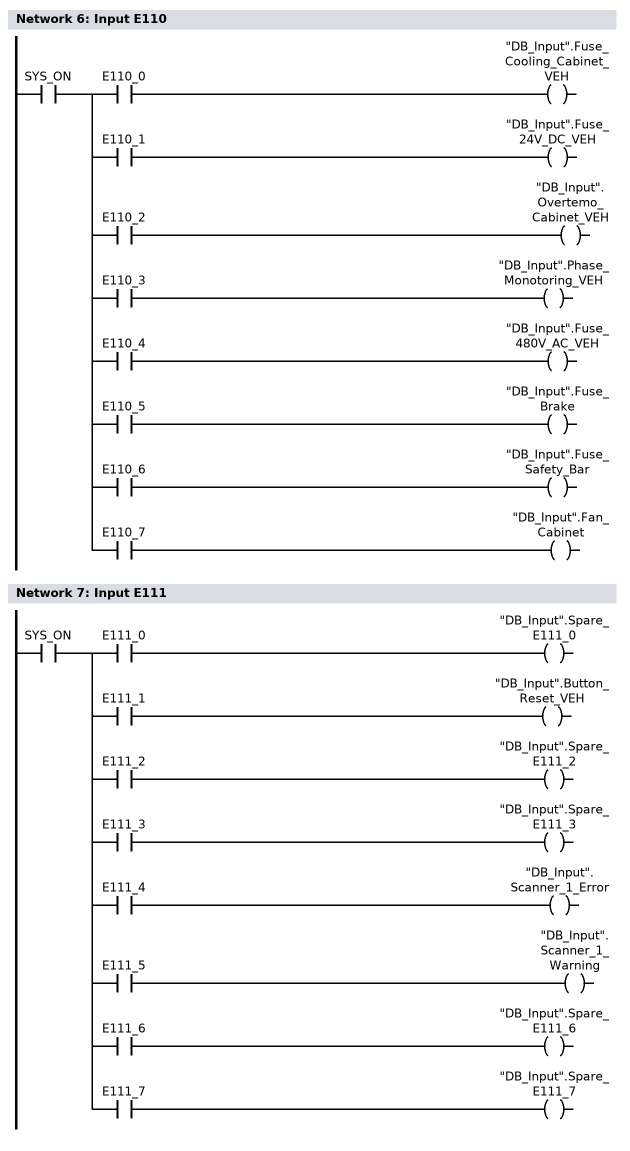
NETWORK
TITLE = Input E110
      A     "SYS_ON";
      =     L 0.0;
      A     L 0.0;
      A     "E110_0";
      =     "DB_Input".Fuse_Cooling_Cabinet_VEH;
      A     L 0.0;
      A     "E110_1";
      =     "DB_Input".Fuse_24V_DC_VEH;
      A     L 0.0;
      A     "E110_2";
      =     "DB_Input".Overtemo_Cabinet_VEH;
      A     L 0.0;
      A     "E110_3";
      =     "DB_Input".Phase_Monotoring_VEH;
      A     L 0.0;
      A     "E110_4";
      =     "DB_Input".Fuse_480V_AC_VEH;
      A     L 0.0;
      A     "E110_5";
      =     "DB_Input".Fuse_Brake;
      A     L 0.0;
      A     "E110_6";
      =     "DB_Input".Fuse_Safety_Bar;
      A     L 0.0;
      A     "E110_7";
      =     "DB_Input".Fan_Cabinet;
NETWORK
TITLE = Input E111
      A     "SYS_ON";
      =     L 0.0;
      A     L 0.0;
      A     "E111_0";
      =     "DB_Input".Spare_E111_0;
      A     L 0.0;
      A     "E111_1";
      =     "DB_Input".Button_Reset_VEH;
      A     L 0.0;
      A     "E111_2";
      =     "DB_Input".Spare_E111_2;
      A     L 0.0;
      A     "E111_3";
      =     "DB_Input".Spare_E111_3;
      A     L 0.0;
      A     "E111_4";
      =     "DB_Input".Scanner_1_Error;
      A     L 0.0;
      A     "E111_5";
      =     "DB_Input".Scanner_1_Warning;
      A     L 0.0;
      A     "E111_6";
      =     "DB_Input".Spare_E111_6;
      A     L 0.0;
      A     "E111_7";
      =     "DB_Input".Spare_E111_7;
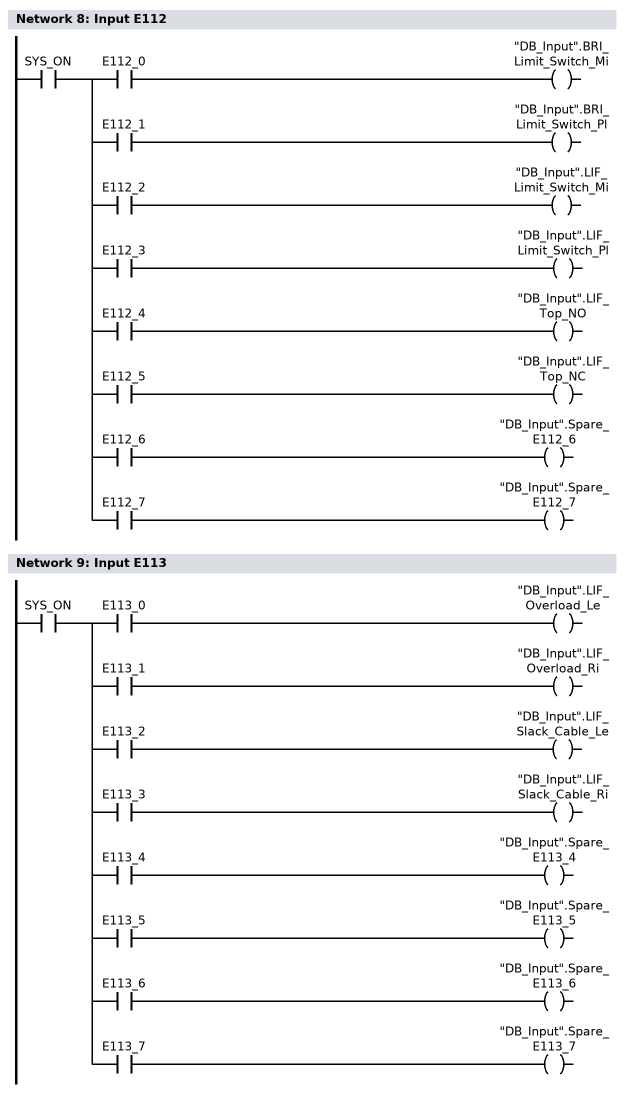
NETWORK
TITLE = Input E112
      A     "SYS_ON";
      =     L 0.0;
      A     L 0.0;
      A     "E112_0";
      =     "DB_Input".BRI_Limit_Switch_Mi;
      A     L 0.0;
      A     "E112_1";
      =     "DB_Input".BRI_Limit_Switch_Pl;
      A     L 0.0;
      A     "E112_2";
      =     "DB_Input".LIF_Limit_Switch_Mi;
      A     L 0.0;
      A     "E112_3";
      =     "DB_Input".LIF_Limit_Switch_Pl;
      A     L 0.0;
      A     "E112_4";
      =     "DB_Input".LIF_Top_NO;
      A     L 0.0;
      A     "E112_5";
      =     "DB_Input".LIF_Top_NC;
      A     L 0.0;
      A     "E112_6";
      =     "DB_Input".Spare_E112_6;
      A     L 0.0;
      A     "E112_7";
      =     "DB_Input".Spare_E112_7;
NETWORK
TITLE = Input E113
      A     "SYS_ON";
      =     L 0.0;
      A     L 0.0;
      A     "E113_0";
      =     "DB_Input".LIF_Overload_Le;
      A     L 0.0;
      A     "E113_1";
      =     "DB_Input".LIF_Overload_Ri;
      A     L 0.0;
      A     "E113_2";
      =     "DB_Input".LIF_Slack_Cable_Le;
      A     L 0.0;
      A     "E113_3";
      =     "DB_Input".LIF_Slack_Cable_Ri;
      A     L 0.0;
      A     "E113_4";
      =     "DB_Input".Spare_E113_4;
      A     L 0.0;
      A     "E113_5";
      =     "DB_Input".Spare_E113_5;
      A     L 0.0;
      A     "E113_6";
      =     "DB_Input".Spare_E113_6;
      A     L 0.0;
      A     "E113_7";
      =     "DB_Input".Spare_E113_7;
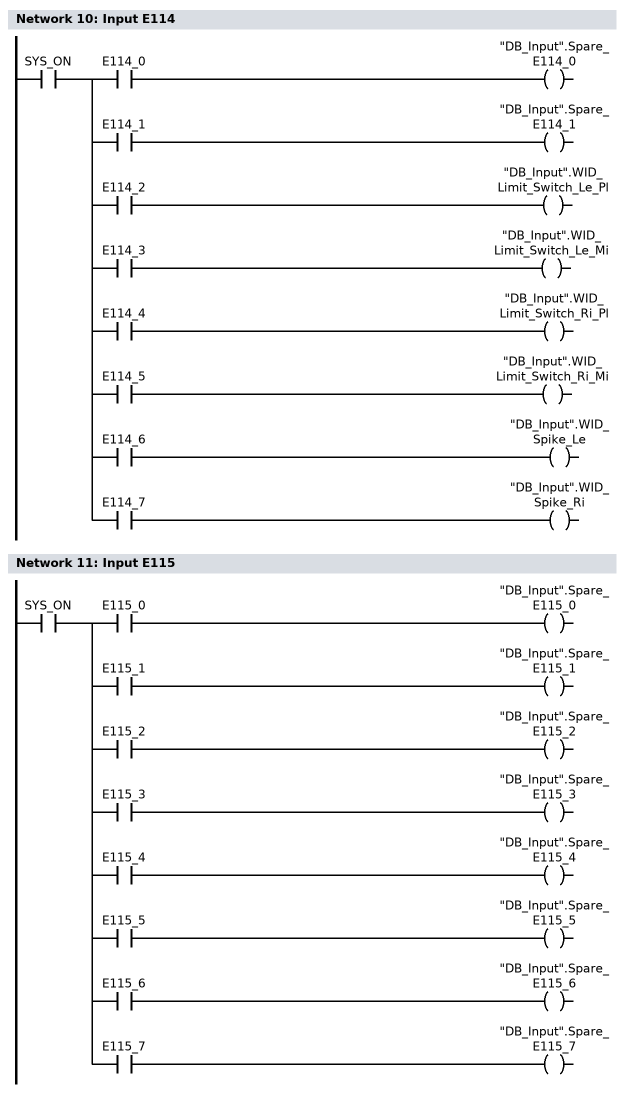
NETWORK
TITLE = Input E114
      A     "SYS_ON";
      =     L 0.0;
      A     L 0.0;
      A     "E114_0";
      =     "DB_Input".Spare_E114_0;
      A     L 0.0;
      A     "E114_1";
      =     "DB_Input".Spare_E114_1;
      A     L 0.0;
      A     "E114_2";
      =     "DB_Input".WID_Limit_Switch_Le_Pl;
      A     L 0.0;
      A     "E114_3";
      =     "DB_Input".WID_Limit_Switch_Le_Mi;
      A     L 0.0;
      A     "E114_4";
      =     "DB_Input".WID_Limit_Switch_Ri_Pl;
      A     L 0.0;
      A     "E114_5";
      =     "DB_Input".WID_Limit_Switch_Ri_Mi;
      A     L 0.0;
      A     "E114_6";
      =     "DB_Input".WID_Spike_Le;
      A     L 0.0;
      A     "E114_7";
      =     "DB_Input".WID_Spike_Ri;
NETWORK
TITLE = Input E115
      A     "SYS_ON";
      =     L 0.0;
      A     L 0.0;
      A     "E115_0";
      =     "DB_Input".Spare_E115_0;
      A     L 0.0;
      A     "E115_1";
      =     "DB_Input".Spare_E115_1;
      A     L 0.0;
      A     "E115_2";
      =     "DB_Input".Spare_E115_2;
      A     L 0.0;
      A     "E115_3";
      =     "DB_Input".Spare_E115_3;
      A     L 0.0;
      A     "E115_4";
      =     "DB_Input".Spare_E115_4;
      A     L 0.0;
      A     "E115_5";
      =     "DB_Input".Spare_E115_5;
      A     L 0.0;
      A     "E115_6";
      =     "DB_Input".Spare_E115_6;
      A     L 0.0;
      A     "E115_7";
      =     "DB_Input".Spare_E115_7;
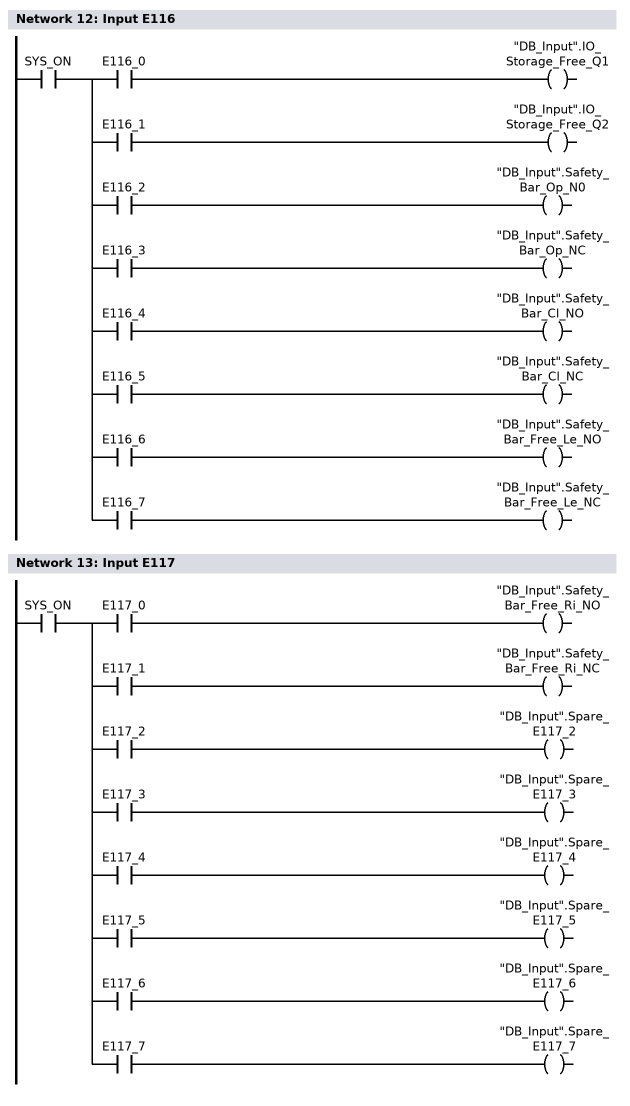
NETWORK
TITLE = Input E116
      A     "SYS_ON";
      =     L 0.0;
      A     L 0.0;
      A     "E116_0";
      =     "DB_Input".IO_Storage_Free_Q1;
      A     L 0.0;
      A     "E116_1";
      =     "DB_Input".IO_Storage_Free_Q2;
      A     L 0.0;
      A     "E116_2";
      =     "DB_Input".Safety_Bar_Op_N0;
      A     L 0.0;
      A     "E116_3";
      =     "DB_Input".Safety_Bar_Op_NC;
      A     L 0.0;
      A     "E116_4";
      =     "DB_Input".Safety_Bar_Cl_NO;
      A     L 0.0;
      A     "E116_5";
      =     "DB_Input".Safety_Bar_Cl_NC;
      A     L 0.0;
      A     "E116_6";
      =     "DB_Input".Safety_Bar_Free_Le_NO;
      A     L 0.0;
      A     "E116_7";
      =     "DB_Input".Safety_Bar_Free_Le_NC;
NETWORK
TITLE = Input E117
      A     "SYS_ON";
      =     L 0.0;
      A     L 0.0;
      A     "E117_0";
      =     "DB_Input".Safety_Bar_Free_Ri_NO;
      A     L 0.0;
      A     "E117_1";
      =     "DB_Input".Safety_Bar_Free_Ri_NC;
      A     L 0.0;
      A     "E117_2";
      =     "DB_Input".Spare_E117_2;
      A     L 0.0;
      A     "E117_3";
      =     "DB_Input".Spare_E117_3;
      A     L 0.0;
      A     "E117_4";
      =     "DB_Input".Spare_E117_4;
      A     L 0.0;
      A     "E117_5";
      =     "DB_Input".Spare_E117_5;
      A     L 0.0;
      A     "E117_6";
      =     "DB_Input".Spare_E117_6;
      A     L 0.0;
      A     "E117_7";
      =     "DB_Input".Spare_E117_7;
END_FUNCTION

FUNCTION "FC_Output" : VOID	// FC 1010
AUTHOR : Broecker
VERSION : 0.1
BEGIN
NETWORK
TITLE =
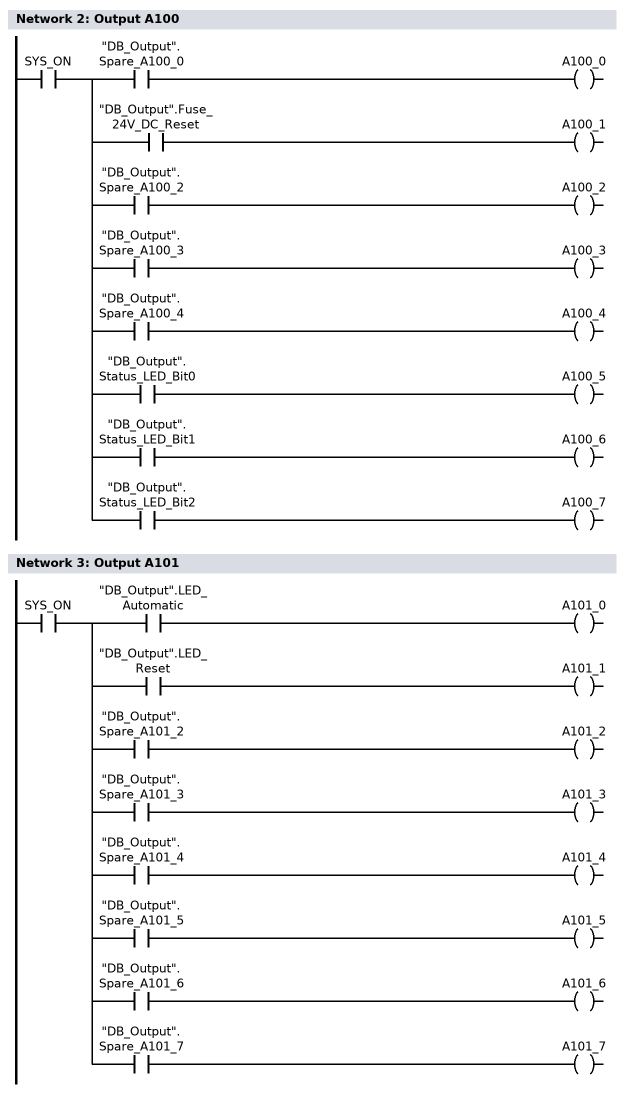
NETWORK
TITLE = Output A100
      A     "SYS_ON";
      =     L 0.0;
      A     L 0.0;
      A     "DB_Output".Spare_A100_0;
      =     "A100_0";
      A     L 0.0;
      A     "DB_Output".Fuse_24V_DC_Reset;
      =     "A100_1";
      A     L 0.0;
      A     "DB_Output".Spare_A100_2;
      =     "A100_2";
      A     L 0.0;
      A     "DB_Output".Spare_A100_3;
      =     "A100_3";
      A     L 0.0;
      A     "DB_Output".Spare_A100_4;
      =     "A100_4";
      A     L 0.0;
      A     "DB_Output".Status_LED_Bit0;
      =     "A100_5";
      A     L 0.0;
      A     "DB_Output".Status_LED_Bit1;
      =     "A100_6";
      A     L 0.0;
      A     "DB_Output".Status_LED_Bit2;
      =     "A100_7";
NETWORK
TITLE = Output A101
      A     "SYS_ON";
      =     L 0.0;
      A     L 0.0;
      A     "DB_Output".LED_Automatic;
      =     "A101_0";
      A     L 0.0;
      A     "DB_Output".LED_Reset;
      =     "A101_1";
      A     L 0.0;
      A     "DB_Output".Spare_A101_2;
      =     "A101_2";
      A     L 0.0;
      A     "DB_Output".Spare_A101_3;
      =     "A101_3";
      A     L 0.0;
      A     "DB_Output".Spare_A101_4;
      =     "A101_4";
      A     L 0.0;
      A     "DB_Output".Spare_A101_5;
      =     "A101_5";
      A     L 0.0;
      A     "DB_Output".Spare_A101_6;
      =     "A101_6";
      A     L 0.0;
      A     "DB_Output".Spare_A101_7;
      =     "A101_7";
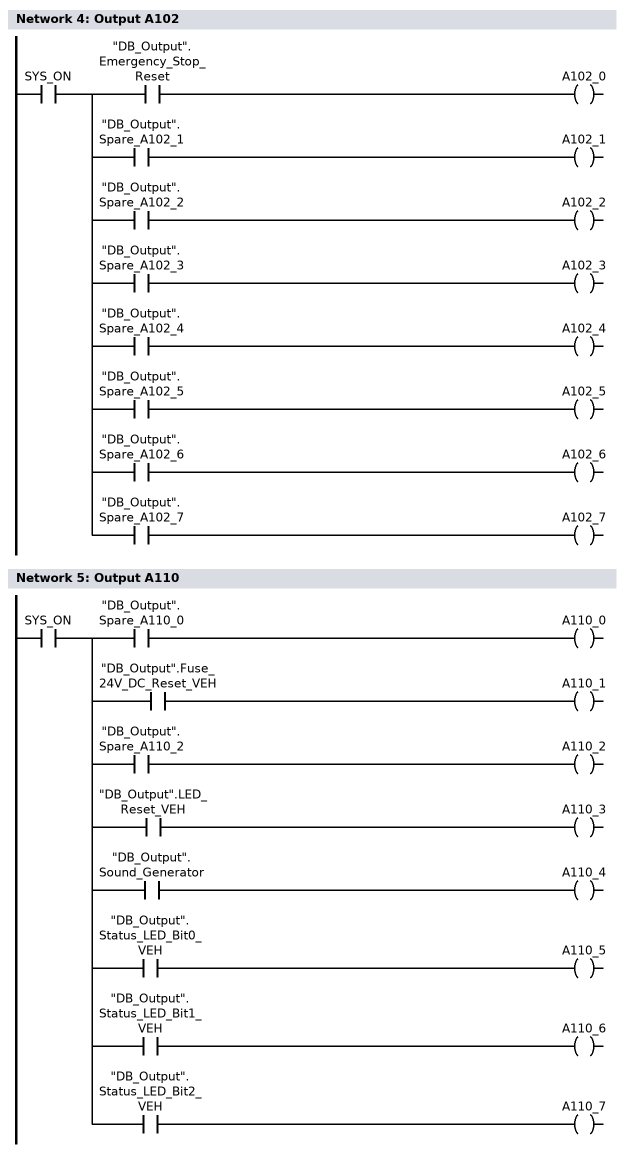
NETWORK
TITLE = Output A102
      A     "SYS_ON";
      =     L 0.0;
      A     L 0.0;
      A     "DB_Output".Emergency_Stop_Reset;
      =     "A102_0";
      A     L 0.0;
      A     "DB_Output".Spare_A102_1;
      =     "A102_1";
      A     L 0.0;
      A     "DB_Output".Spare_A102_2;
      =     "A102_2";
      A     L 0.0;
      A     "DB_Output".Spare_A102_3;
      =     "A102_3";
      A     L 0.0;
      A     "DB_Output".Spare_A102_4;
      =     "A102_4";
      A     L 0.0;
      A     "DB_Output".Spare_A102_5;
      =     "A102_5";
      A     L 0.0;
      A     "DB_Output".Spare_A102_6;
      =     "A102_6";
      A     L 0.0;
      A     "DB_Output".Spare_A102_7;
      =     "A102_7";
NETWORK
TITLE = Output A110
      A     "SYS_ON";
      =     L 0.0;
      A     L 0.0;
      A     "DB_Output".Spare_A110_0;
      =     "A110_0";
      A     L 0.0;
      A     "DB_Output".Fuse_24V_DC_Reset_VEH;
      =     "A110_1";
      A     L 0.0;
      A     "DB_Output".Spare_A110_2;
      =     "A110_2";
      A     L 0.0;
      A     "DB_Output".LED_Reset_VEH;
      =     "A110_3";
      A     L 0.0;
      A     "DB_Output".Sound_Generator;
      =     "A110_4";
      A     L 0.0;
      A     "DB_Output".Status_LED_Bit0_VEH;
      =     "A110_5";
      A     L 0.0;
      A     "DB_Output".Status_LED_Bit1_VEH;
      =     "A110_6";
      A     L 0.0;
      A     "DB_Output".Status_LED_Bit2_VEH;
      =     "A110_7";
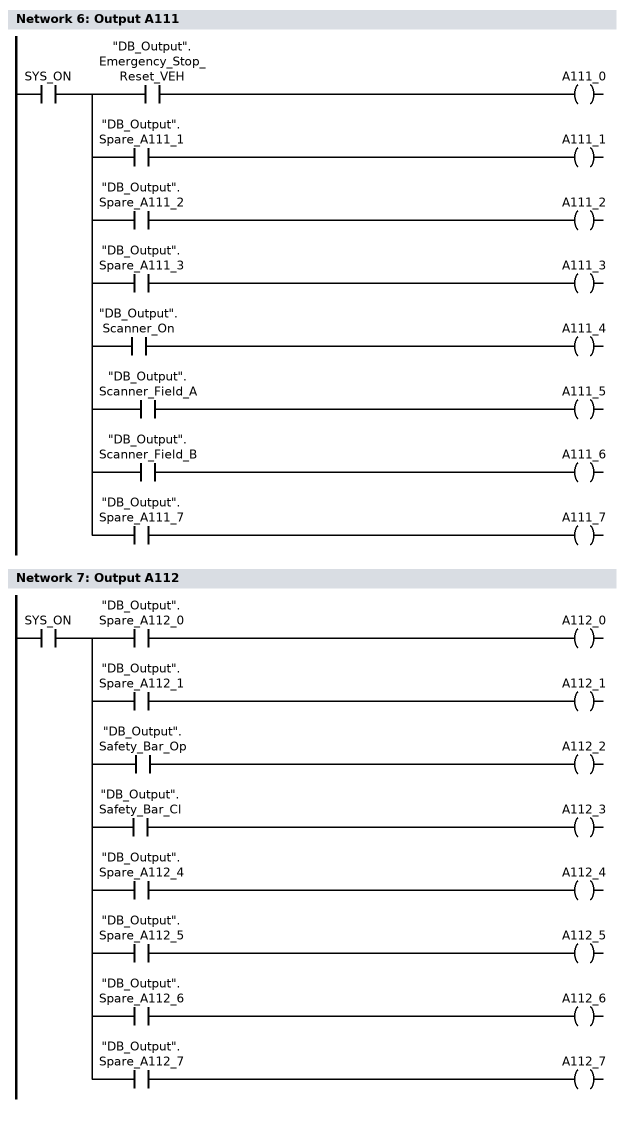
NETWORK
TITLE = Output A111
      A     "SYS_ON";
      =     L 0.0;
      A     L 0.0;
      A     "DB_Output".Emergency_Stop_Reset_VEH;
      =     "A111_0";
      A     L 0.0;
      A     "DB_Output".Spare_A111_1;
      =     "A111_1";
      A     L 0.0;
      A     "DB_Output".Spare_A111_2;
      =     "A111_2";
      A     L 0.0;
      A     "DB_Output".Spare_A111_3;
      =     "A111_3";
      A     L 0.0;
      A     "DB_Output".Scanner_On;
      =     "A111_4";
      A     L 0.0;
      A     "DB_Output".Scanner_Field_A;
      =     "A111_5";
      A     L 0.0;
      A     "DB_Output".Scanner_Field_B;
      =     "A111_6";
      A     L 0.0;
      A     "DB_Output".Spare_A111_7;
      =     "A111_7";
NETWORK
TITLE = Output A112
      A     "SYS_ON";
      =     L 0.0;
      A     L 0.0;
      A     "DB_Output".Spare_A112_0;
      =     "A112_0";
      A     L 0.0;
      A     "DB_Output".Spare_A112_1;
      =     "A112_1";
      A     L 0.0;
      A     "DB_Output".Safety_Bar_Op;
      =     "A112_2";
      A     L 0.0;
      A     "DB_Output".Safety_Bar_Cl;
      =     "A112_3";
      A     L 0.0;
      A     "DB_Output".Spare_A112_4;
      =     "A112_4";
      A     L 0.0;
      A     "DB_Output".Spare_A112_5;
      =     "A112_5";
      A     L 0.0;
      A     "DB_Output".Spare_A112_6;
      =     "A112_6";
      A     L 0.0;
      A     "DB_Output".Spare_A112_7;
      =     "A112_7";
END_FUNCTION

DATA_BLOCK "DBS_Input"	// DB 100
AUTHOR : Broecker
VERSION : 0.1
  STRUCT
   IN_ESTOP_Extern_CH1 : BOOL ;
   IN_ESTOP_Extern_CH2 : BOOL ;
   Spare_E020_2 : BOOL ;
   Spare_E020_3 : BOOL ;
   Spare_E020_4 : BOOL ;
   Spare_E020_5 : BOOL ;
   Spare_E020_6 : BOOL ;
   Spare_E020_7 : BOOL ;
   ESTOP_CH1 : BOOL ;
   ESTOP_CH2 : BOOL ;
   Spare_E025_2 : BOOL ;
   Spare_E025_3 : BOOL ;
   Automatic_Mode_CH1 : BOOL ;
   Automatic_Mode_CH2 : BOOL ;
   Service_Mode_CH1 : BOOL ;
   Service_Mode_CH2 : BOOL ;
   Spare_E030_0 : BOOL ;
   Spare_E030_1 : BOOL ;
   Spare_E030_2 : BOOL ;
   Spare_E030_3 : BOOL ;
   Spare_E030_4 : BOOL ;
   Spare_E030_5 : BOOL ;
   Spare_E030_6 : BOOL ;
   Spare_E030_7 : BOOL ;
   Spare_E035_0 : BOOL ;
   Spare_E035_1 : BOOL ;
   Spare_E035_2 : BOOL ;
   Spare_E035_3 : BOOL ;
   Spare_E035_4 : BOOL ;
   Spare_E035_5 : BOOL ;
   Spare_E035_6 : BOOL ;
   Spare_E035_7 : BOOL ;
   Spare_E040_0 : BOOL ;
   Spare_E040_1 : BOOL ;
   Spare_E040_2 : BOOL ;
   Spare_E040_3 : BOOL ;
   Spare_E040_4 : BOOL ;
   Spare_E040_5 : BOOL ;
   Spare_E040_6 : BOOL ;
   Spare_E040_7 : BOOL ;
   Spare_E045_0 : BOOL ;
   Spare_E045_1 : BOOL ;
   Spare_E045_2 : BOOL ;
   Spare_E045_3 : BOOL ;
   Spare_E045_4 : BOOL ;
   Spare_E045_5 : BOOL ;
   Spare_E045_6 : BOOL ;
   Spare_E045_7 : BOOL ;
   Spare_E050_0 : BOOL ;
   IN_BRI_Fast_Stop : BOOL ;
   IN_LIF_Fast_Stop : BOOL ;
   IN_WID_Fast_Stop : BOOL ;
   Spare_E050_4 : BOOL ;
   Spare_E050_5 : BOOL ;
   Spare_E050_6 : BOOL ;
   Spare_E050_7 : BOOL ;
   Spare_E055_0 : BOOL ;
   IN_ESTOP_CH12 : BOOL ;
   LIF_Overload_NC : BOOL ;
   LIF_Slack_Cable_NC : BOOL ;
   Spare_E055_4 : BOOL ;
   Spare_E055_5 : BOOL ;
   Spare_E055_6 : BOOL ;
   Spare_E055_7 : BOOL ;
   WID_Le_RoSw_On_CH1 : BOOL ;
   WID_Le_RoSw_On_CH2 : BOOL ;
   WID_Le_RoSw_Off_CH1 : BOOL ;
   WID_Le_RoSw_Off_CH2 : BOOL ;
   WID_Le_PaSw_On_CH1 : BOOL ;
   WID_Le_PaSw_On_CH2 : BOOL ;
   WID_Le_PaSw_Off_CH1 : BOOL ;
   WID_Le_PaSw_Off_CH2 : BOOL ;
   WID_Ri_RoSw_On_CH1 : BOOL ;
   WID_Ri_RoSw_On_CH2 : BOOL ;
   WID_Ri_RoSw_Off_CH1 : BOOL ;
   WID_Ri_RoSw_Off_CH2 : BOOL ;
   WID_Ri_PaSw_On_CH1 : BOOL ;
   WID_Ri_PaSw_On_CH2 : BOOL ;
   WID_Ri_PaSw_Off_CH1 : BOOL ;
   WID_Ri_PaSw_Off_CH2 : BOOL ;
   Safety_Bar_Cl_CH1 : BOOL ;
   Safety_Bar_Cl_CH2 : BOOL ;
   Scanner_1_OSSD1 : BOOL ;
   Scanner_1_OSSD2 : BOOL ;
   Spare_E070_4 : BOOL ;
   Spare_E070_5 : BOOL ;
   Spare_E070_6 : BOOL ;
   Spare_E070_7 : BOOL ;
   Spare_E075_0 : BOOL ;
   Spare_E075_1 : BOOL ;
   Spare_E075_2 : BOOL ;
   Spare_E075_3 : BOOL ;
   No_ESTOP : BOOL ;
   No_Overtemp_Brake : BOOL ;
   Bypass_Mode_CH1 : BOOL ;
   Bypass_Mode_CH2 : BOOL ;
  END_STRUCT ;	
BEGIN
END_DATA_BLOCK

DATA_BLOCK "DBS_Output"	// DB 110
AUTHOR : Broecker
VERSION : 0.1
  STRUCT
   OUT_ESTOP_Extern_CH1 : BOOL ;
   OUT_ESTOP_Extern_CH2 : BOOL ;
   Spare_A020_2 : BOOL ;
   Spare_A020_3 : BOOL ;
   Spare_A020_4 : BOOL ;
   Spare_A020_5 : BOOL ;
   Spare_A020_6 : BOOL ;
   Spare_A020_7 : BOOL ;
   Spare_A025_0 : BOOL ;
   Spare_A025_1 : BOOL ;
   Spare_A025_2 : BOOL ;
   Spare_A025_3 : BOOL ;
   Spare_A025_4 : BOOL ;
   Spare_A025_5 : BOOL ;
   Spare_A025_6 : BOOL ;
   Spare_A025_7 : BOOL ;
   Spare_A030_0 : BOOL ;
   Spare_A030_1 : BOOL ;
   Spare_A030_2 : BOOL ;
   Spare_A030_3 : BOOL ;
   Spare_A030_4 : BOOL ;
   Spare_A030_5 : BOOL ;
   Spare_A030_6 : BOOL ;
   Spare_A030_7 : BOOL ;
   Spare_A035_0 : BOOL ;
   Spare_A035_1 : BOOL ;
   Spare_A035_2 : BOOL ;
   Spare_A035_3 : BOOL ;
   Spare_A035_4 : BOOL ;
   Spare_A035_5 : BOOL ;
   Spare_A035_6 : BOOL ;
   Spare_A035_7 : BOOL ;
   Spare_A040_0 : BOOL ;
   Spare_A040_1 : BOOL ;
   Spare_A040_2 : BOOL ;
   Spare_A040_3 : BOOL ;
   Spare_A040_4 : BOOL ;
   Spare_A040_5 : BOOL ;
   Spare_A040_6 : BOOL ;
   Spare_A040_7 : BOOL ;
   Spare_A045_0 : BOOL ;
   Spare_A045_1 : BOOL ;
   Spare_A045_2 : BOOL ;
   Spare_A045_3 : BOOL ;
   Spare_A045_4 : BOOL ;
   Spare_A045_5 : BOOL ;
   Spare_A045_6 : BOOL ;
   Spare_A045_7 : BOOL ;
   Spare_A050_0 : BOOL ;
   OUT_BRI_Fast_Stop : BOOL ;
   OUT_LIF_Fast_Stop : BOOL ;
   OUT_WID_Fast_Stop : BOOL ;
   Spare_A050_4 : BOOL ;
   Spare_A050_5 : BOOL ;
   Spare_A050_6 : BOOL ;
   Spare_A050_7 : BOOL ;
   Spare_A055_0 : BOOL ;
   Spare_A055_1 : BOOL ;
   OUT_ESTOP_CH1 : BOOL ;
   OUT_ESTOP_CH2 : BOOL ;
   Spare_A055_4 : BOOL ;
   Spare_A055_5 : BOOL ;
   Spare_A055_6 : BOOL ;
   Spare_A055_7 : BOOL ;
   Spare_A060_0 : BOOL ;
   Spare_A060_1 : BOOL ;
   Spare_A060_2 : BOOL ;
   Spare_A060_3 : BOOL ;
   Spare_A060_4 : BOOL ;
   Spare_A060_5 : BOOL ;
   Spare_A060_6 : BOOL ;
   Spare_A060_7 : BOOL ;
   Spare_A065_0 : BOOL ;
   Spare_A065_1 : BOOL ;
   Spare_A065_2 : BOOL ;
   Spare_A065_3 : BOOL ;
   Spare_A065_4 : BOOL ;
   Spare_A065_5 : BOOL ;
   Spare_A065_6 : BOOL ;
   Spare_A065_7 : BOOL ;
   Spare_A070_0 : BOOL ;
   Spare_A070_1 : BOOL ;
   Spare_A070_2 : BOOL ;
   Spare_A070_3 : BOOL ;
   Spare_A070_4 : BOOL ;
   Spare_A070_5 : BOOL ;
   Spare_A070_6 : BOOL ;
   Spare_A070_7 : BOOL ;
   Spare_A075_0 : BOOL ;
   Spare_A075_1 : BOOL ;
   Spare_A075_2 : BOOL ;
   Spare_A075_3 : BOOL ;
   Spare_A075_4 : BOOL ;
   Spare_A075_5 : BOOL ;
   Spare_A075_6 : BOOL ;
   Spare_A075_7 : BOOL ;
  END_STRUCT ;	
BEGIN
END_DATA_BLOCK

DATA_BLOCK "DB_Input"	// DB 1000
VERSION : 0.1
  STRUCT
   Spare_E100_0 : BOOL ;
   Fuse_24V_DC : BOOL ;
   Overtemp_Cabinet : BOOL ;
   Phase_Monotoring : BOOL ;
   Spare_E100_4 : BOOL ;
   Spare_E100_5 : BOOL ;
   Spare_E100_6 : BOOL ;
   Spare_E100_7 : BOOL ;
   Button_Automatic : BOOL ;
   Button_Reset : BOOL ;
   Spare_E101_2 : BOOL ;
   Spare_E101_3 : BOOL ;
   Spare_E101_4 : BOOL ;
   Button_Emergency_Stop_1 : BOOL ;
   Button_Emergency_Stop_2 : BOOL ;
   Button_Emergency_Stop_3 : BOOL ;
   Spare_E102_0 : BOOL ;
   Spare_E102_1 : BOOL ;
   Spare_E102_2 : BOOL ;
   Spare_E102_3 : BOOL ;
   Spare_E102_4 : BOOL ;
   Spare_E102_5 : BOOL ;
   Spare_E102_6 : BOOL ;
   Spare_E102_7 : BOOL ;
   Spare_E103_0 : BOOL ;
   Spare_E103_1 : BOOL ;
   Spare_E103_2 : BOOL ;
   Spare_E103_3 : BOOL ;
   Spare_E103_4 : BOOL ;
   Spare_E103_5 : BOOL ;
   Spare_E103_6 : BOOL ;
   Spare_E103_7 : BOOL ;
   Spare_E104_0 : BOOL ;
   Spare_E104_1 : BOOL ;
   Spare_E104_2 : BOOL ;
   Spare_E104_3 : BOOL ;
   Spare_E104_4 : BOOL ;
   Spare_E104_5 : BOOL ;
   Spare_E104_6 : BOOL ;
   Spare_E104_7 : BOOL ;
   Spare_E105_0 : BOOL ;
   Spare_E105_1 : BOOL ;
   Spare_E105_2 : BOOL ;
   Spare_E105_3 : BOOL ;
   Spare_E105_4 : BOOL ;
   Spare_E105_5 : BOOL ;
   Spare_E105_6 : BOOL ;
   Spare_E105_7 : BOOL ;
   Spare_E106_0 : BOOL ;
   Spare_E106_1 : BOOL ;
   Spare_E106_2 : BOOL ;
   Spare_E106_3 : BOOL ;
   Spare_E106_4 : BOOL ;
   Spare_E106_5 : BOOL ;
   Spare_E106_6 : BOOL ;
   Spare_E106_7 : BOOL ;
   Spare_E107_0 : BOOL ;
   Spare_E107_1 : BOOL ;
   Spare_E107_2 : BOOL ;
   Spare_E107_3 : BOOL ;
   Spare_E107_4 : BOOL ;
   Spare_E107_5 : BOOL ;
   Spare_E107_6 : BOOL ;
   Spare_E107_7 : BOOL ;
   Spare_E108_0 : BOOL ;
   Spare_E108_1 : BOOL ;
   Spare_E108_2 : BOOL ;
   Spare_E108_3 : BOOL ;
   Spare_E108_4 : BOOL ;
   Spare_E108_5 : BOOL ;
   Spare_E108_6 : BOOL ;
   Spare_E108_7 : BOOL ;
   Spare_E109_0 : BOOL ;
   Spare_E109_1 : BOOL ;
   Spare_E109_2 : BOOL ;
   Spare_E109_3 : BOOL ;
   Spare_E109_4 : BOOL ;
   Spare_E109_5 : BOOL ;
   Spare_E109_6 : BOOL ;
   Spare_E109_7 : BOOL ;
   Fuse_Cooling_Cabinet_VEH : BOOL ;
   Fuse_24V_DC_VEH : BOOL ;
   Overtemo_Cabinet_VEH : BOOL ;
   Phase_Monotoring_VEH : BOOL ;
   Fuse_480V_AC_VEH : BOOL ;
   Fuse_Brake : BOOL ;
   Fuse_Safety_Bar : BOOL ;
   Fan_Cabinet : BOOL ;
   Spare_E111_0 : BOOL ;
   Button_Reset_VEH : BOOL ;
   Spare_E111_2 : BOOL ;
   Spare_E111_3 : BOOL ;
   Scanner_1_Error : BOOL ;
   Scanner_1_Warning : BOOL ;
   Spare_E111_6 : BOOL ;
   Spare_E111_7 : BOOL ;
   BRI_Limit_Switch_Mi : BOOL ;
   BRI_Limit_Switch_Pl : BOOL ;
   LIF_Limit_Switch_Mi : BOOL ;
   LIF_Limit_Switch_Pl : BOOL ;
   LIF_Top_NO : BOOL ;
   LIF_Top_NC : BOOL ;
   Spare_E112_6 : BOOL ;
   Spare_E112_7 : BOOL ;
   LIF_Overload_Le : BOOL ;
   LIF_Overload_Ri : BOOL ;
   LIF_Slack_Cable_Le : BOOL ;
   LIF_Slack_Cable_Ri : BOOL ;
   Spare_E113_4 : BOOL ;
   Spare_E113_5 : BOOL ;
   Spare_E113_6 : BOOL ;
   Spare_E113_7 : BOOL ;
   Spare_E114_0 : BOOL ;
   Spare_E114_1 : BOOL ;
   WID_Limit_Switch_Le_Pl : BOOL ;
   WID_Limit_Switch_Le_Mi : BOOL ;
   WID_Limit_Switch_Ri_Pl : BOOL ;
   WID_Limit_Switch_Ri_Mi : BOOL ;
   WID_Spike_Le : BOOL ;
   WID_Spike_Ri : BOOL ;
   Spare_E115_0 : BOOL ;
   Spare_E115_1 : BOOL ;
   Spare_E115_2 : BOOL ;
   Spare_E115_3 : BOOL ;
   Spare_E115_4 : BOOL ;
   Spare_E115_5 : BOOL ;
   Spare_E115_6 : BOOL ;
   Spare_E115_7 : BOOL ;
   IO_Storage_Free_Q1 : BOOL ;
   IO_Storage_Free_Q2 : BOOL ;
   Safety_Bar_Op_N0 : BOOL ;
   Safety_Bar_Op_NC : BOOL ;
   Safety_Bar_Cl_NO : BOOL ;
   Safety_Bar_Cl_NC : BOOL ;
   Safety_Bar_Free_Le_NO : BOOL ;
   Safety_Bar_Free_Le_NC : BOOL ;
   Safety_Bar_Free_Ri_NO : BOOL ;
   Safety_Bar_Free_Ri_NC : BOOL ;
   Spare_E117_2 : BOOL ;
   Spare_E117_3 : BOOL ;
   Spare_E117_4 : BOOL ;
   Spare_E117_5 : BOOL ;
   Spare_E117_6 : BOOL ;
   Spare_E117_7 : BOOL ;
   Spare_E118_0 : BOOL ;
   Spare_E118_1 : BOOL ;
   Spare_E118_2 : BOOL ;
   Spare_E118_3 : BOOL ;
   Spare_E118_4 : BOOL ;
   Spare_E118_5 : BOOL ;
   Spare_E118_6 : BOOL ;
   Spare_E118_7 : BOOL ;
  END_STRUCT ;	
BEGIN
END_DATA_BLOCK

